// TIA Portal V17 export
// export: Created 2024-09-02T12:50:15.8804122Z, ExportSetting WithDefaults, DisplayName Totally Integrated Automation Portal, DisplayVersion V17, DisplayName TIA Portal Openness, DisplayVersion V17, DisplayName TIA Portal Version Control Interface, DisplayVersion V17, DisplayName STEP 7 Professional, DisplayVersion V17, DisplayName STEP 7 Safety, DisplayVersion V17, DisplayName WinCC Professional, DisplayVersion V17
FUNCTION "AnwFC_ZP_FunctionsSelection_OP70" : Void   // FC254, LAD
TITLE = function selections / Funktionsanwahlen
{ S7_Optimized_Access := 'TRUE' }
AUTHOR : OlegFuehrus
FAMILY : BA
NAME : BA
VERSION : 0.1
// stored: AutoNumber true, IsIECCheckEnabled false, SetENOAutomatically false, UDAEnableTagReadback false
   VAR_TEMP
      t_VKE0 : Bool;
      t_VKE1 : Bool;
      t_Enable_left : Bool;
      t_Enable_right : Bool;
      t_Fault : Bool;
      t_Function_left : Bool;
      t_Function_right : Bool;
      t_Line : Int;
      tBA_mode : Int;
   END_VAR
   VAR_TEMP   // added for the SCL form of the ladder/FBD networks
      _w1 : Bool;
      _w2 : Bool;
      _w3 : Bool;
      _w4 : Bool;
      _w5 : Bool;
   END_VAR
BEGIN

REGION Network 1: INIT
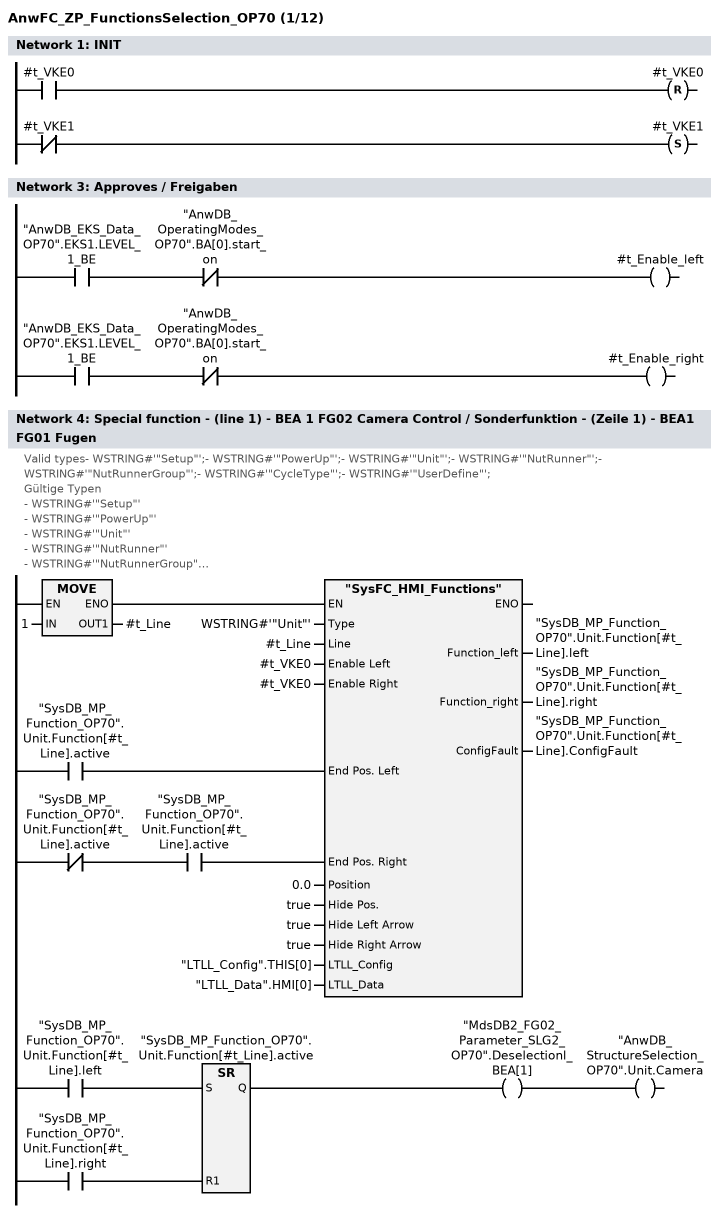
   RUNG wire#powerrail
      Contact( #t_VKE0 )
      R_Coil( #t_VKE0 )
   END_RUNG
   RUNG wire#powerrail
      I_Contact( #t_VKE1 )
      S_Coil( #t_VKE1 )
   END_RUNG
   // the same network as SCL:
   IF #t_VKE0 THEN #t_VKE0 := FALSE; END_IF;
   IF NOT #t_VKE1 THEN #t_VKE1 := TRUE; END_IF;
END_REGION

REGION Network 2: ######## UNIT ######### / ############ UNIT ############
END_REGION

REGION Network 3: Approves / Freigaben
   RUNG wire#powerrail
      Contact( "AnwDB_EKS_Data_OP70".EKS1.LEVEL_1_BE )
      I_Contact( "AnwDB_OperatingModes_OP70".BA[0].start_on )
      Coil( #t_Enable_left )
   END_RUNG
   RUNG wire#powerrail
      Contact( "AnwDB_EKS_Data_OP70".EKS1.LEVEL_1_BE )
      I_Contact( "AnwDB_OperatingModes_OP70".BA[0].start_on )
      Coil( #t_Enable_right )
   END_RUNG
   // the same network as SCL:
   #t_Enable_left := "AnwDB_EKS_Data_OP70".EKS1.LEVEL_1_BE AND NOT "AnwDB_OperatingModes_OP70".BA[0].start_on;
   #t_Enable_right := "AnwDB_EKS_Data_OP70".EKS1.LEVEL_1_BE AND NOT "AnwDB_OperatingModes_OP70".BA[0].start_on;
END_REGION

REGION Network 4: Special function - (line 1) - BEA 1 FG02 Camera Control / Sonderfunktion - (Zeile 1) - BEA1 FG01 Fugen
   // Valid types- WSTRING#'"Setup"';- WSTRING#'"PowerUp"';- WSTRING#'"Unit"';- WSTRING#'"NutRunner"';- WSTRING#'"NutRunnerGroup"';- WSTRING#'"CycleType"';- WSTRING#'"UserDefine"';
   // Gültige Typen
   // - WSTRING#'"Setup"'
   // - WSTRING#'"PowerUp"'
   // - WSTRING#'"Unit"'
   // - WSTRING#'"NutRunner"'
   // - WSTRING#'"NutRunnerGroup"'
   // - WSTRING#'"CycleType"'
   // - WSTRING#'"UserDefine"'
   RUNG wire#powerrail
      Move(in := 1, out1 => #t_Line)
      "SysFC_HMI_Functions"("End Pos. Left" := wire#w1, "End Pos. Right" := wire#w2, "Type" := WSTRING#'"Unit"', Line := #t_Line, "Enable Left" := #t_VKE0, "Enable Right" := #t_VKE0, Position := 0.0, "Hide Pos." := true, "Hide Left Arrow" := true, "Hide Right Arrow" := true, LTLL_Config := "LTLL_Config".THIS[0], LTLL_Data := "LTLL_Data".HMI[0], Function_left => "SysDB_MP_Function_OP70".Unit.Function[#t_Line].left, Function_right => "SysDB_MP_Function_OP70".Unit.Function[#t_Line].right, ConfigFault => "SysDB_MP_Function_OP70".Unit.Function[#t_Line].ConfigFault)
   END_RUNG
   RUNG wire#powerrail
      Contact( "SysDB_MP_Function_OP70".Unit.Function[#t_Line].active )
   END_RUNG wire#w1
   RUNG wire#powerrail
      I_Contact( "SysDB_MP_Function_OP70".Unit.Function[#t_Line].active )
      Contact( "SysDB_MP_Function_OP70".Unit.Function[#t_Line].active )
   END_RUNG wire#w2
   RUNG wire#powerrail
      Contact( "SysDB_MP_Function_OP70".Unit.Function[#t_Line].left )
      S_SR(operand := "SysDB_MP_Function_OP70".Unit.Function[#t_Line].active, r1 := wire#w3)
      Coil( "MdsDB2_FG02_Parameter_SLG2_OP70".Deselectionl_BEA[1] )
      Coil( "AnwDB_StructureSelection_OP70".Unit.Camera )
   END_RUNG
   RUNG wire#powerrail
      Contact( "SysDB_MP_Function_OP70".Unit.Function[#t_Line].right )
   END_RUNG wire#w3
   // the same network as SCL:
   #t_Line := 1;
   "SysFC_HMI_Functions"("Type" := WSTRING#'"Unit"',
                         Line := #t_Line,
                         "Enable Left" := #t_VKE0,
                         "Enable Right" := #t_VKE0,
                         "End Pos. Left" := "SysDB_MP_Function_OP70".Unit.Function[#t_Line].active,
                         "End Pos. Right" := NOT "SysDB_MP_Function_OP70".Unit.Function[#t_Line].active AND "SysDB_MP_Function_OP70".Unit.Function[#t_Line].active,
                         Position := 0.0,
                         "Hide Pos." := true,
                         "Hide Left Arrow" := true,
                         "Hide Right Arrow" := true,
                         LTLL_Config := "LTLL_Config".THIS[0],
                         LTLL_Data := "LTLL_Data".HMI[0],
                         Function_left => "SysDB_MP_Function_OP70".Unit.Function[#t_Line].left,
                         Function_right => "SysDB_MP_Function_OP70".Unit.Function[#t_Line].right,
                         ConfigFault => "SysDB_MP_Function_OP70".Unit.Function[#t_Line].ConfigFault);
   #_w1 := "SysDB_MP_Function_OP70".Unit.Function[#t_Line].right;
   IF "SysDB_MP_Function_OP70".Unit.Function[#t_Line].left THEN
       "SysDB_MP_Function_OP70".Unit.Function[#t_Line].active := TRUE;   // SR flip-flop
   END_IF;
   IF #_w1 THEN "SysDB_MP_Function_OP70".Unit.Function[#t_Line].active := FALSE; END_IF;
   "MdsDB2_FG02_Parameter_SLG2_OP70".Deselectionl_BEA[1] := "SysDB_MP_Function_OP70".Unit.Function[#t_Line].active;
   "AnwDB_StructureSelection_OP70".Unit.Camera := "SysDB_MP_Function_OP70".Unit.Function[#t_Line].active;
END_REGION

REGION Network 5: Special function - (line 2) - BEA 2 FG02 Replace plate / Sonderfunktion - (Zeile 1) - BEA1 FG01 Fugen
   // Valid types- WSTRING#'"Setup"';- WSTRING#'"PowerUp"';- WSTRING#'"Unit"';- WSTRING#'"NutRunner"';- WSTRING#'"NutRunnerGroup"';- WSTRING#'"CycleType"';- WSTRING#'"UserDefine"';
   // Gültige Typen
   // - WSTRING#'"Setup"'
   // - WSTRING#'"PowerUp"'
   // - WSTRING#'"Unit"'
   // - WSTRING#'"NutRunner"'
   // - WSTRING#'"NutRunnerGroup"'
   // - WSTRING#'"CycleType"'
   // - WSTRING#'"UserDefine"'
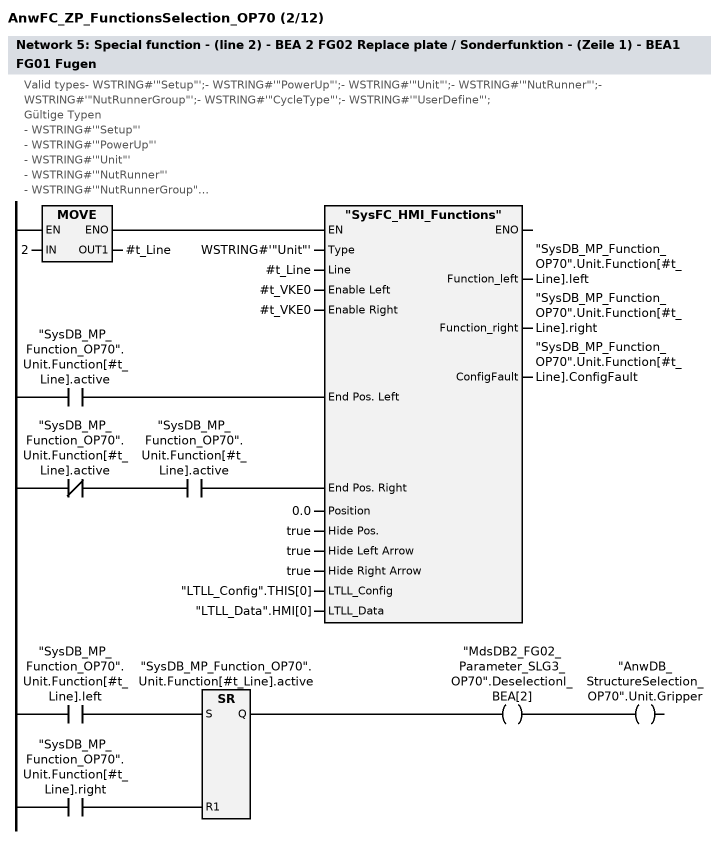
   RUNG wire#powerrail
      Move(in := 2, out1 => #t_Line)
      "SysFC_HMI_Functions"("End Pos. Left" := wire#w1, "End Pos. Right" := wire#w2, "Type" := WSTRING#'"Unit"', Line := #t_Line, "Enable Left" := #t_VKE0, "Enable Right" := #t_VKE0, Position := 0.0, "Hide Pos." := true, "Hide Left Arrow" := true, "Hide Right Arrow" := true, LTLL_Config := "LTLL_Config".THIS[0], LTLL_Data := "LTLL_Data".HMI[0], Function_left => "SysDB_MP_Function_OP70".Unit.Function[#t_Line].left, Function_right => "SysDB_MP_Function_OP70".Unit.Function[#t_Line].right, ConfigFault => "SysDB_MP_Function_OP70".Unit.Function[#t_Line].ConfigFault)
   END_RUNG
   RUNG wire#powerrail
      Contact( "SysDB_MP_Function_OP70".Unit.Function[#t_Line].active )
   END_RUNG wire#w1
   RUNG wire#powerrail
      I_Contact( "SysDB_MP_Function_OP70".Unit.Function[#t_Line].active )
      Contact( "SysDB_MP_Function_OP70".Unit.Function[#t_Line].active )
   END_RUNG wire#w2
   RUNG wire#powerrail
      Contact( "SysDB_MP_Function_OP70".Unit.Function[#t_Line].left )
      S_SR(operand := "SysDB_MP_Function_OP70".Unit.Function[#t_Line].active, r1 := wire#w3)
      Coil( "MdsDB2_FG02_Parameter_SLG3_OP70".Deselectionl_BEA[2] )
      Coil( "AnwDB_StructureSelection_OP70".Unit.Gripper )
   END_RUNG
   RUNG wire#powerrail
      Contact( "SysDB_MP_Function_OP70".Unit.Function[#t_Line].right )
   END_RUNG wire#w3
   // the same network as SCL:
   #t_Line := 2;
   "SysFC_HMI_Functions"("Type" := WSTRING#'"Unit"',
                         Line := #t_Line,
                         "Enable Left" := #t_VKE0,
                         "Enable Right" := #t_VKE0,
                         "End Pos. Left" := "SysDB_MP_Function_OP70".Unit.Function[#t_Line].active,
                         "End Pos. Right" := NOT "SysDB_MP_Function_OP70".Unit.Function[#t_Line].active AND "SysDB_MP_Function_OP70".Unit.Function[#t_Line].active,
                         Position := 0.0,
                         "Hide Pos." := true,
                         "Hide Left Arrow" := true,
                         "Hide Right Arrow" := true,
                         LTLL_Config := "LTLL_Config".THIS[0],
                         LTLL_Data := "LTLL_Data".HMI[0],
                         Function_left => "SysDB_MP_Function_OP70".Unit.Function[#t_Line].left,
                         Function_right => "SysDB_MP_Function_OP70".Unit.Function[#t_Line].right,
                         ConfigFault => "SysDB_MP_Function_OP70".Unit.Function[#t_Line].ConfigFault);
   #_w1 := "SysDB_MP_Function_OP70".Unit.Function[#t_Line].right;
   IF "SysDB_MP_Function_OP70".Unit.Function[#t_Line].left THEN
       "SysDB_MP_Function_OP70".Unit.Function[#t_Line].active := TRUE;   // SR flip-flop
   END_IF;
   IF #_w1 THEN "SysDB_MP_Function_OP70".Unit.Function[#t_Line].active := FALSE; END_IF;
   "MdsDB2_FG02_Parameter_SLG3_OP70".Deselectionl_BEA[2] := "SysDB_MP_Function_OP70".Unit.Function[#t_Line].active;
   "AnwDB_StructureSelection_OP70".Unit.Gripper := "SysDB_MP_Function_OP70".Unit.Function[#t_Line].active;
END_REGION

REGION Network 6: Special function - (line 3) - BEA 3 FG02 Screwdriver / Sonderfunktion - (Zeile 1) - BEA1 FG01 Fugen
   // Valid types- WSTRING#'"Setup"';- WSTRING#'"PowerUp"';- WSTRING#'"Unit"';- WSTRING#'"NutRunner"';- WSTRING#'"NutRunnerGroup"';- WSTRING#'"CycleType"';- WSTRING#'"UserDefine"';
   // Gültige Typen
   // - WSTRING#'"Setup"'
   // - WSTRING#'"PowerUp"'
   // - WSTRING#'"Unit"'
   // - WSTRING#'"NutRunner"'
   // - WSTRING#'"NutRunnerGroup"'
   // - WSTRING#'"CycleType"'
   // - WSTRING#'"UserDefine"'
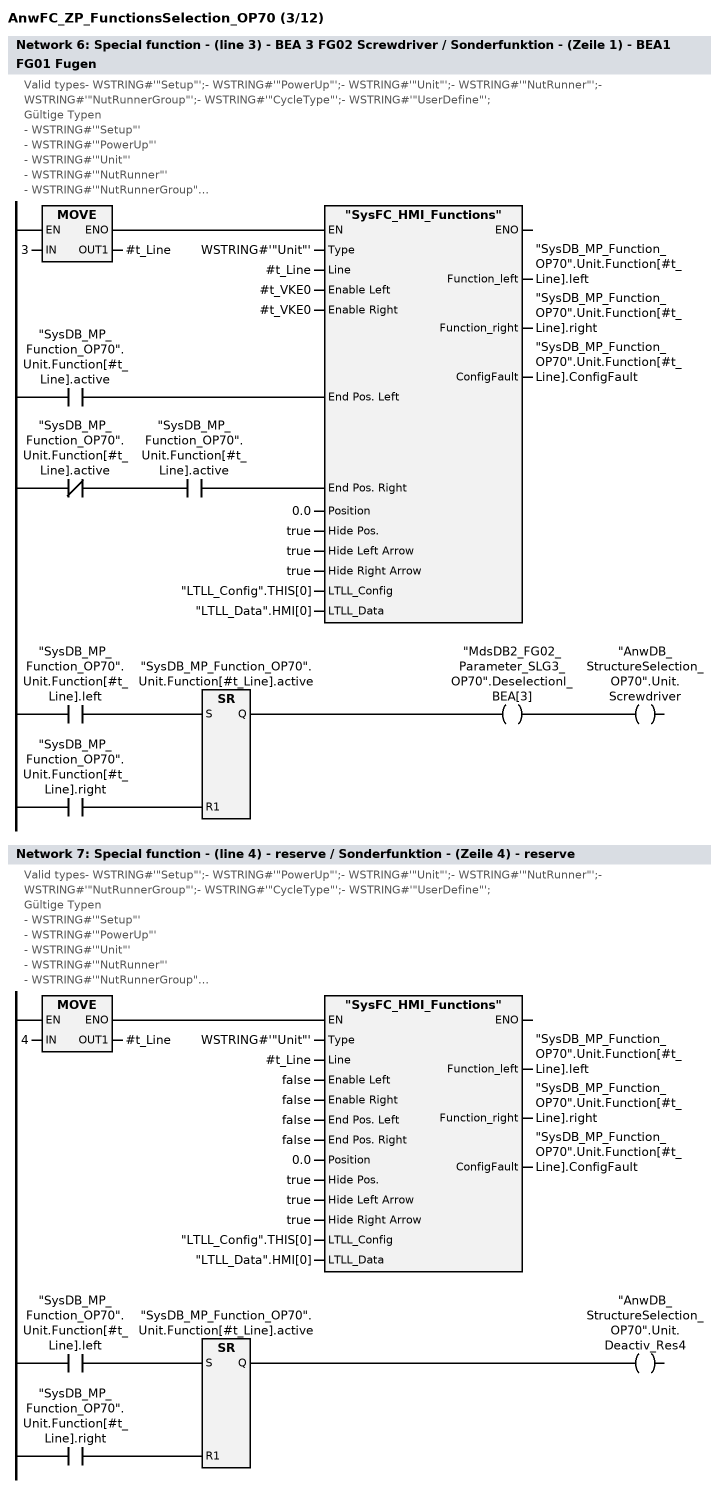
   RUNG wire#powerrail
      Move(in := 3, out1 => #t_Line)
      "SysFC_HMI_Functions"("End Pos. Left" := wire#w1, "End Pos. Right" := wire#w2, "Type" := WSTRING#'"Unit"', Line := #t_Line, "Enable Left" := #t_VKE0, "Enable Right" := #t_VKE0, Position := 0.0, "Hide Pos." := true, "Hide Left Arrow" := true, "Hide Right Arrow" := true, LTLL_Config := "LTLL_Config".THIS[0], LTLL_Data := "LTLL_Data".HMI[0], Function_left => "SysDB_MP_Function_OP70".Unit.Function[#t_Line].left, Function_right => "SysDB_MP_Function_OP70".Unit.Function[#t_Line].right, ConfigFault => "SysDB_MP_Function_OP70".Unit.Function[#t_Line].ConfigFault)
   END_RUNG
   RUNG wire#powerrail
      Contact( "SysDB_MP_Function_OP70".Unit.Function[#t_Line].active )
   END_RUNG wire#w1
   RUNG wire#powerrail
      I_Contact( "SysDB_MP_Function_OP70".Unit.Function[#t_Line].active )
      Contact( "SysDB_MP_Function_OP70".Unit.Function[#t_Line].active )
   END_RUNG wire#w2
   RUNG wire#powerrail
      Contact( "SysDB_MP_Function_OP70".Unit.Function[#t_Line].left )
      S_SR(operand := "SysDB_MP_Function_OP70".Unit.Function[#t_Line].active, r1 := wire#w3)
      Coil( "MdsDB2_FG02_Parameter_SLG3_OP70".Deselectionl_BEA[3] )
      Coil( "AnwDB_StructureSelection_OP70".Unit.Screwdriver )
   END_RUNG
   RUNG wire#powerrail
      Contact( "SysDB_MP_Function_OP70".Unit.Function[#t_Line].right )
   END_RUNG wire#w3
   // the same network as SCL:
   #t_Line := 3;
   "SysFC_HMI_Functions"("Type" := WSTRING#'"Unit"',
                         Line := #t_Line,
                         "Enable Left" := #t_VKE0,
                         "Enable Right" := #t_VKE0,
                         "End Pos. Left" := "SysDB_MP_Function_OP70".Unit.Function[#t_Line].active,
                         "End Pos. Right" := NOT "SysDB_MP_Function_OP70".Unit.Function[#t_Line].active AND "SysDB_MP_Function_OP70".Unit.Function[#t_Line].active,
                         Position := 0.0,
                         "Hide Pos." := true,
                         "Hide Left Arrow" := true,
                         "Hide Right Arrow" := true,
                         LTLL_Config := "LTLL_Config".THIS[0],
                         LTLL_Data := "LTLL_Data".HMI[0],
                         Function_left => "SysDB_MP_Function_OP70".Unit.Function[#t_Line].left,
                         Function_right => "SysDB_MP_Function_OP70".Unit.Function[#t_Line].right,
                         ConfigFault => "SysDB_MP_Function_OP70".Unit.Function[#t_Line].ConfigFault);
   #_w1 := "SysDB_MP_Function_OP70".Unit.Function[#t_Line].right;
   IF "SysDB_MP_Function_OP70".Unit.Function[#t_Line].left THEN
       "SysDB_MP_Function_OP70".Unit.Function[#t_Line].active := TRUE;   // SR flip-flop
   END_IF;
   IF #_w1 THEN "SysDB_MP_Function_OP70".Unit.Function[#t_Line].active := FALSE; END_IF;
   "MdsDB2_FG02_Parameter_SLG3_OP70".Deselectionl_BEA[3] := "SysDB_MP_Function_OP70".Unit.Function[#t_Line].active;
   "AnwDB_StructureSelection_OP70".Unit.Screwdriver := "SysDB_MP_Function_OP70".Unit.Function[#t_Line].active;
END_REGION

REGION Network 7: Special function - (line 4) - reserve / Sonderfunktion - (Zeile 4) - reserve
   // Valid types- WSTRING#'"Setup"';- WSTRING#'"PowerUp"';- WSTRING#'"Unit"';- WSTRING#'"NutRunner"';- WSTRING#'"NutRunnerGroup"';- WSTRING#'"CycleType"';- WSTRING#'"UserDefine"';
   // Gültige Typen
   // - WSTRING#'"Setup"'
   // - WSTRING#'"PowerUp"'
   // - WSTRING#'"Unit"'
   // - WSTRING#'"NutRunner"'
   // - WSTRING#'"NutRunnerGroup"'
   // - WSTRING#'"CycleType"'
   // - WSTRING#'"UserDefine"'
   RUNG wire#powerrail
      Move(in := 4, out1 => #t_Line)
      "SysFC_HMI_Functions"("Type" := WSTRING#'"Unit"', Line := #t_Line, "Enable Left" := false, "Enable Right" := false, "End Pos. Left" := false, "End Pos. Right" := false, Position := 0.0, "Hide Pos." := true, "Hide Left Arrow" := true, "Hide Right Arrow" := true, LTLL_Config := "LTLL_Config".THIS[0], LTLL_Data := "LTLL_Data".HMI[0], Function_left => "SysDB_MP_Function_OP70".Unit.Function[#t_Line].left, Function_right => "SysDB_MP_Function_OP70".Unit.Function[#t_Line].right, ConfigFault => "SysDB_MP_Function_OP70".Unit.Function[#t_Line].ConfigFault)
   END_RUNG
   RUNG wire#powerrail
      Contact( "SysDB_MP_Function_OP70".Unit.Function[#t_Line].left )
      S_SR(operand := "SysDB_MP_Function_OP70".Unit.Function[#t_Line].active, r1 := wire#w1)
      Coil( "AnwDB_StructureSelection_OP70".Unit.Deactiv_Res4 )
   END_RUNG
   RUNG wire#powerrail
      Contact( "SysDB_MP_Function_OP70".Unit.Function[#t_Line].right )
   END_RUNG wire#w1
   // the same network as SCL:
   #t_Line := 4;
   "SysFC_HMI_Functions"("Type" := WSTRING#'"Unit"',
                         Line := #t_Line,
                         "Enable Left" := false,
                         "Enable Right" := false,
                         "End Pos. Left" := false,
                         "End Pos. Right" := false,
                         Position := 0.0,
                         "Hide Pos." := true,
                         "Hide Left Arrow" := true,
                         "Hide Right Arrow" := true,
                         LTLL_Config := "LTLL_Config".THIS[0],
                         LTLL_Data := "LTLL_Data".HMI[0],
                         Function_left => "SysDB_MP_Function_OP70".Unit.Function[#t_Line].left,
                         Function_right => "SysDB_MP_Function_OP70".Unit.Function[#t_Line].right,
                         ConfigFault => "SysDB_MP_Function_OP70".Unit.Function[#t_Line].ConfigFault);
   #_w1 := "SysDB_MP_Function_OP70".Unit.Function[#t_Line].right;
   IF "SysDB_MP_Function_OP70".Unit.Function[#t_Line].left THEN
       "SysDB_MP_Function_OP70".Unit.Function[#t_Line].active := TRUE;   // SR flip-flop
   END_IF;
   IF #_w1 THEN "SysDB_MP_Function_OP70".Unit.Function[#t_Line].active := FALSE; END_IF;
   "AnwDB_StructureSelection_OP70".Unit.Deactiv_Res4 := "SysDB_MP_Function_OP70".Unit.Function[#t_Line].active;
END_REGION

REGION Network 8: Special function - (line 5) - reserve / Sonderfunktion - (Zeile 5) - reserve
   // Valid types- WSTRING#'"Setup"';- WSTRING#'"PowerUp"';- WSTRING#'"Unit"';- WSTRING#'"NutRunner"';- WSTRING#'"NutRunnerGroup"';- WSTRING#'"CycleType"';- WSTRING#'"UserDefine"';
   // Gültige Typen
   // - WSTRING#'"Setup"'
   // - WSTRING#'"PowerUp"'
   // - WSTRING#'"Unit"'
   // - WSTRING#'"NutRunner"'
   // - WSTRING#'"NutRunnerGroup"'
   // - WSTRING#'"CycleType"'
   // - WSTRING#'"UserDefine"'
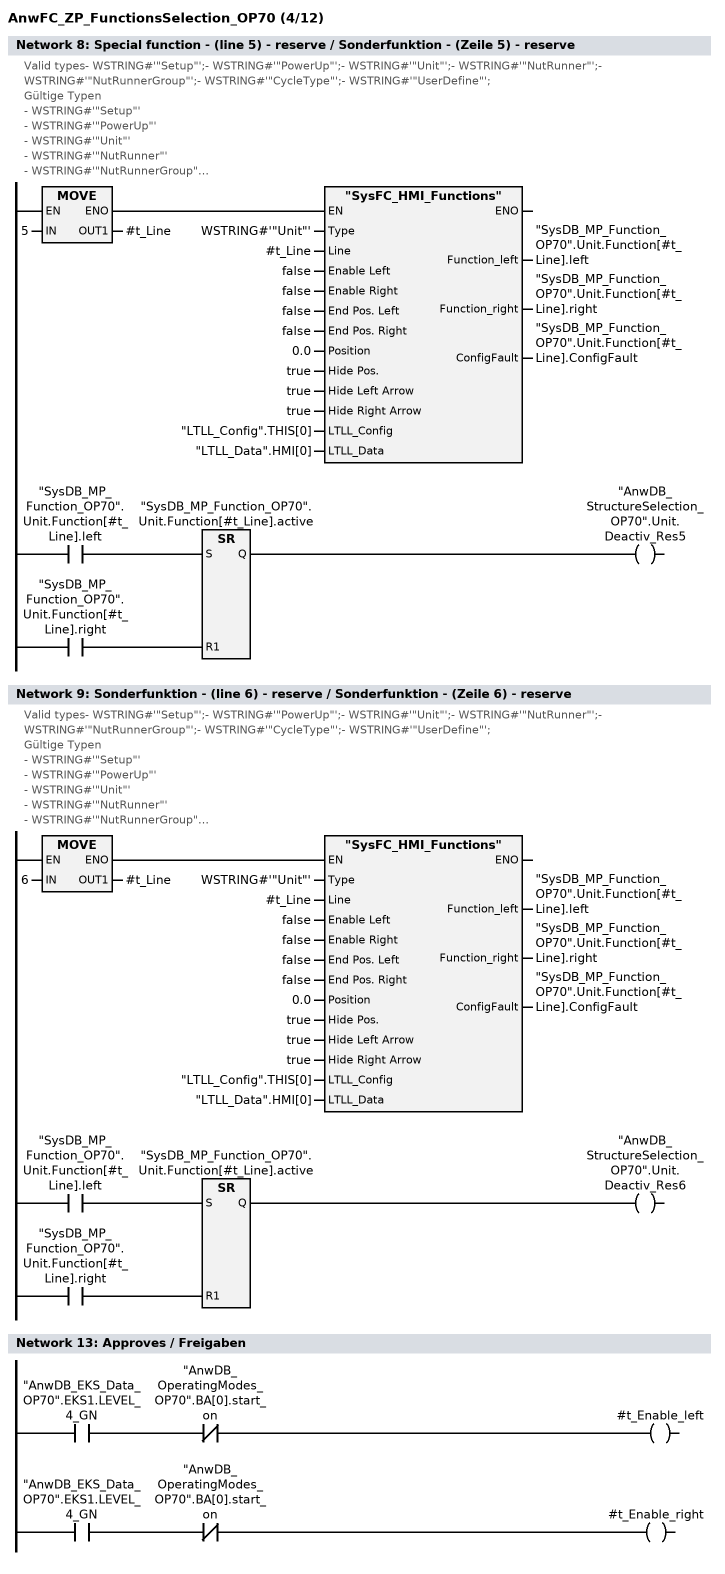
   RUNG wire#powerrail
      Move(in := 5, out1 => #t_Line)
      "SysFC_HMI_Functions"("Type" := WSTRING#'"Unit"', Line := #t_Line, "Enable Left" := false, "Enable Right" := false, "End Pos. Left" := false, "End Pos. Right" := false, Position := 0.0, "Hide Pos." := true, "Hide Left Arrow" := true, "Hide Right Arrow" := true, LTLL_Config := "LTLL_Config".THIS[0], LTLL_Data := "LTLL_Data".HMI[0], Function_left => "SysDB_MP_Function_OP70".Unit.Function[#t_Line].left, Function_right => "SysDB_MP_Function_OP70".Unit.Function[#t_Line].right, ConfigFault => "SysDB_MP_Function_OP70".Unit.Function[#t_Line].ConfigFault)
   END_RUNG
   RUNG wire#powerrail
      Contact( "SysDB_MP_Function_OP70".Unit.Function[#t_Line].left )
      S_SR(operand := "SysDB_MP_Function_OP70".Unit.Function[#t_Line].active, r1 := wire#w1)
      Coil( "AnwDB_StructureSelection_OP70".Unit.Deactiv_Res5 )
   END_RUNG
   RUNG wire#powerrail
      Contact( "SysDB_MP_Function_OP70".Unit.Function[#t_Line].right )
   END_RUNG wire#w1
   // the same network as SCL:
   #t_Line := 5;
   "SysFC_HMI_Functions"("Type" := WSTRING#'"Unit"',
                         Line := #t_Line,
                         "Enable Left" := false,
                         "Enable Right" := false,
                         "End Pos. Left" := false,
                         "End Pos. Right" := false,
                         Position := 0.0,
                         "Hide Pos." := true,
                         "Hide Left Arrow" := true,
                         "Hide Right Arrow" := true,
                         LTLL_Config := "LTLL_Config".THIS[0],
                         LTLL_Data := "LTLL_Data".HMI[0],
                         Function_left => "SysDB_MP_Function_OP70".Unit.Function[#t_Line].left,
                         Function_right => "SysDB_MP_Function_OP70".Unit.Function[#t_Line].right,
                         ConfigFault => "SysDB_MP_Function_OP70".Unit.Function[#t_Line].ConfigFault);
   #_w1 := "SysDB_MP_Function_OP70".Unit.Function[#t_Line].right;
   IF "SysDB_MP_Function_OP70".Unit.Function[#t_Line].left THEN
       "SysDB_MP_Function_OP70".Unit.Function[#t_Line].active := TRUE;   // SR flip-flop
   END_IF;
   IF #_w1 THEN "SysDB_MP_Function_OP70".Unit.Function[#t_Line].active := FALSE; END_IF;
   "AnwDB_StructureSelection_OP70".Unit.Deactiv_Res5 := "SysDB_MP_Function_OP70".Unit.Function[#t_Line].active;
END_REGION

REGION Network 9: Sonderfunktion - (line 6) - reserve / Sonderfunktion - (Zeile 6) - reserve
   // Valid types- WSTRING#'"Setup"';- WSTRING#'"PowerUp"';- WSTRING#'"Unit"';- WSTRING#'"NutRunner"';- WSTRING#'"NutRunnerGroup"';- WSTRING#'"CycleType"';- WSTRING#'"UserDefine"';
   // Gültige Typen
   // - WSTRING#'"Setup"'
   // - WSTRING#'"PowerUp"'
   // - WSTRING#'"Unit"'
   // - WSTRING#'"NutRunner"'
   // - WSTRING#'"NutRunnerGroup"'
   // - WSTRING#'"CycleType"'
   // - WSTRING#'"UserDefine"'
   RUNG wire#powerrail
      Move(in := 6, out1 => #t_Line)
      "SysFC_HMI_Functions"("Type" := WSTRING#'"Unit"', Line := #t_Line, "Enable Left" := false, "Enable Right" := false, "End Pos. Left" := false, "End Pos. Right" := false, Position := 0.0, "Hide Pos." := true, "Hide Left Arrow" := true, "Hide Right Arrow" := true, LTLL_Config := "LTLL_Config".THIS[0], LTLL_Data := "LTLL_Data".HMI[0], Function_left => "SysDB_MP_Function_OP70".Unit.Function[#t_Line].left, Function_right => "SysDB_MP_Function_OP70".Unit.Function[#t_Line].right, ConfigFault => "SysDB_MP_Function_OP70".Unit.Function[#t_Line].ConfigFault)
   END_RUNG
   RUNG wire#powerrail
      Contact( "SysDB_MP_Function_OP70".Unit.Function[#t_Line].left )
      S_SR(operand := "SysDB_MP_Function_OP70".Unit.Function[#t_Line].active, r1 := wire#w1)
      Coil( "AnwDB_StructureSelection_OP70".Unit.Deactiv_Res6 )
   END_RUNG
   RUNG wire#powerrail
      Contact( "SysDB_MP_Function_OP70".Unit.Function[#t_Line].right )
   END_RUNG wire#w1
   // the same network as SCL:
   #t_Line := 6;
   "SysFC_HMI_Functions"("Type" := WSTRING#'"Unit"',
                         Line := #t_Line,
                         "Enable Left" := false,
                         "Enable Right" := false,
                         "End Pos. Left" := false,
                         "End Pos. Right" := false,
                         Position := 0.0,
                         "Hide Pos." := true,
                         "Hide Left Arrow" := true,
                         "Hide Right Arrow" := true,
                         LTLL_Config := "LTLL_Config".THIS[0],
                         LTLL_Data := "LTLL_Data".HMI[0],
                         Function_left => "SysDB_MP_Function_OP70".Unit.Function[#t_Line].left,
                         Function_right => "SysDB_MP_Function_OP70".Unit.Function[#t_Line].right,
                         ConfigFault => "SysDB_MP_Function_OP70".Unit.Function[#t_Line].ConfigFault);
   #_w1 := "SysDB_MP_Function_OP70".Unit.Function[#t_Line].right;
   IF "SysDB_MP_Function_OP70".Unit.Function[#t_Line].left THEN
       "SysDB_MP_Function_OP70".Unit.Function[#t_Line].active := TRUE;   // SR flip-flop
   END_IF;
   IF #_w1 THEN "SysDB_MP_Function_OP70".Unit.Function[#t_Line].active := FALSE; END_IF;
   "AnwDB_StructureSelection_OP70".Unit.Deactiv_Res6 := "SysDB_MP_Function_OP70".Unit.Function[#t_Line].active;
END_REGION

REGION Network 10: ######## NUT RUNNER ######### / ############ NUT RUNNER ############
END_REGION

REGION Network 11: ######## NUT RUNNER GROUP ######### / ############ NUT RUNNER GROUP ############
END_REGION

REGION Network 12: ######## CYCLE TYPE ######### / ############ CYCLE TYPE ############
END_REGION

REGION Network 13: Approves / Freigaben
   RUNG wire#powerrail
      Contact( "AnwDB_EKS_Data_OP70".EKS1.LEVEL_4_GN )
      I_Contact( "AnwDB_OperatingModes_OP70".BA[0].start_on )
      Coil( #t_Enable_left )
   END_RUNG
   RUNG wire#powerrail
      Contact( "AnwDB_EKS_Data_OP70".EKS1.LEVEL_4_GN )
      I_Contact( "AnwDB_OperatingModes_OP70".BA[0].start_on )
      Coil( #t_Enable_right )
   END_RUNG
   // the same network as SCL:
   #t_Enable_left := "AnwDB_EKS_Data_OP70".EKS1.LEVEL_4_GN AND NOT "AnwDB_OperatingModes_OP70".BA[0].start_on;
   #t_Enable_right := "AnwDB_EKS_Data_OP70".EKS1.LEVEL_4_GN AND NOT "AnwDB_OperatingModes_OP70".BA[0].start_on;
END_REGION

REGION Network 14: CycleType - (line 1) - Single step mode / CycleType - (Zeile 1) - Einzelschritt
   // Valid types- WSTRING#'"Setup"';- WSTRING#'"PowerUp"';- WSTRING#'"Unit"';- WSTRING#'"NutRunner"';- WSTRING#'"NutRunnerGroup"';- WSTRING#'"CycleType"';- WSTRING#'"UserDefine"';
   // Gültige Typen
   // - WSTRING#'"Setup"'
   // - WSTRING#'"PowerUp"'
   // - WSTRING#'"Unit"'
   // - WSTRING#'"NutRunner"'
   // - WSTRING#'"NutRunnerGroup"'
   // - WSTRING#'"CycleType"'
   // - WSTRING#'"UserDefine"'
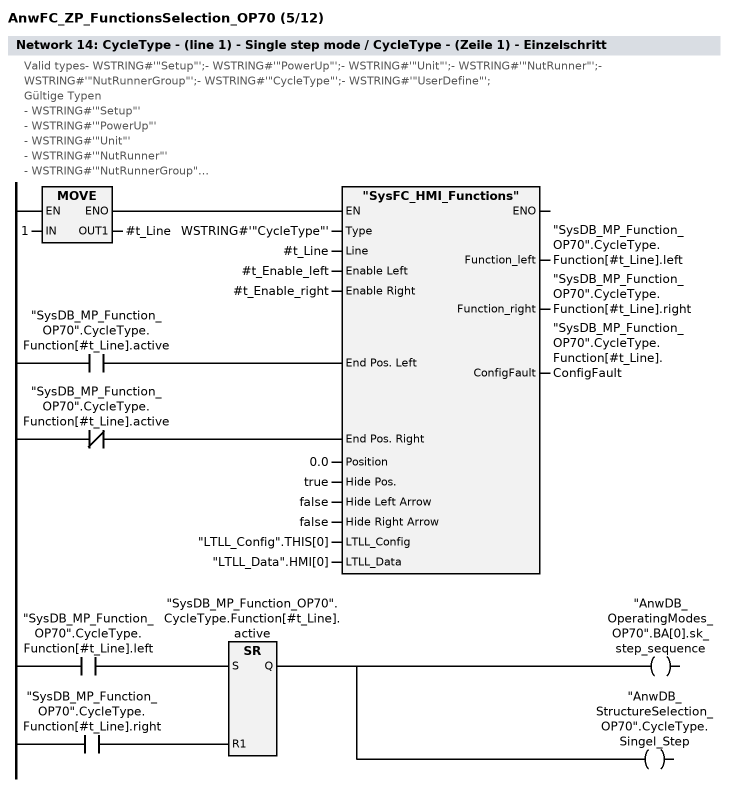
   RUNG wire#powerrail
      Move(in := 1, out1 => #t_Line)
      "SysFC_HMI_Functions"("End Pos. Left" := wire#w1, "End Pos. Right" := wire#w2, "Type" := WSTRING#'"CycleType"', Line := #t_Line, "Enable Left" := #t_Enable_left, "Enable Right" := #t_Enable_right, Position := 0.0, "Hide Pos." := true, "Hide Left Arrow" := false, "Hide Right Arrow" := false, LTLL_Config := "LTLL_Config".THIS[0], LTLL_Data := "LTLL_Data".HMI[0], Function_left => "SysDB_MP_Function_OP70".CycleType.Function[#t_Line].left, Function_right => "SysDB_MP_Function_OP70".CycleType.Function[#t_Line].right, ConfigFault => "SysDB_MP_Function_OP70".CycleType.Function[#t_Line].ConfigFault)
   END_RUNG
   RUNG wire#powerrail
      Contact( "SysDB_MP_Function_OP70".CycleType.Function[#t_Line].active )
   END_RUNG wire#w1
   RUNG wire#powerrail
      I_Contact( "SysDB_MP_Function_OP70".CycleType.Function[#t_Line].active )
   END_RUNG wire#w2
   RUNG wire#powerrail
      Contact( "SysDB_MP_Function_OP70".CycleType.Function[#t_Line].left )
      S_SR(operand := "SysDB_MP_Function_OP70".CycleType.Function[#t_Line].active, r1 := wire#w3)
      wire#w4
      Coil( "AnwDB_OperatingModes_OP70".BA[0].sk_step_sequence )
   END_RUNG
   RUNG wire#powerrail
      Contact( "SysDB_MP_Function_OP70".CycleType.Function[#t_Line].right )
   END_RUNG wire#w3
   RUNG wire#w4
      Coil( "AnwDB_StructureSelection_OP70".CycleType.Singel_Step )
   END_RUNG
   // the same network as SCL:
   #t_Line := 1;
   "SysFC_HMI_Functions"("Type" := WSTRING#'"CycleType"',
                         Line := #t_Line,
                         "Enable Left" := #t_Enable_left,
                         "Enable Right" := #t_Enable_right,
                         "End Pos. Left" := "SysDB_MP_Function_OP70".CycleType.Function[#t_Line].active,
                         "End Pos. Right" := NOT "SysDB_MP_Function_OP70".CycleType.Function[#t_Line].active,
                         Position := 0.0,
                         "Hide Pos." := true,
                         "Hide Left Arrow" := false,
                         "Hide Right Arrow" := false,
                         LTLL_Config := "LTLL_Config".THIS[0],
                         LTLL_Data := "LTLL_Data".HMI[0],
                         Function_left => "SysDB_MP_Function_OP70".CycleType.Function[#t_Line].left,
                         Function_right => "SysDB_MP_Function_OP70".CycleType.Function[#t_Line].right,
                         ConfigFault => "SysDB_MP_Function_OP70".CycleType.Function[#t_Line].ConfigFault);
   #_w1 := "SysDB_MP_Function_OP70".CycleType.Function[#t_Line].right;
   IF "SysDB_MP_Function_OP70".CycleType.Function[#t_Line].left THEN
       "SysDB_MP_Function_OP70".CycleType.Function[#t_Line].active := TRUE;   // SR flip-flop
   END_IF;
   IF #_w1 THEN "SysDB_MP_Function_OP70".CycleType.Function[#t_Line].active := FALSE; END_IF;
   "AnwDB_OperatingModes_OP70".BA[0].sk_step_sequence := "SysDB_MP_Function_OP70".CycleType.Function[#t_Line].active;
   "AnwDB_StructureSelection_OP70".CycleType.Singel_Step := "SysDB_MP_Function_OP70".CycleType.Function[#t_Line].active;
END_REGION

REGION Network 15: CycleType - (line 2) - Service / CycleType - (Zeile 2) - Service
   // Valid types- WSTRING#'"Setup"';- WSTRING#'"PowerUp"';- WSTRING#'"Unit"';- WSTRING#'"NutRunner"';- WSTRING#'"NutRunnerGroup"';- WSTRING#'"CycleType"';- WSTRING#'"UserDefine"';
   // Gültige Typen
   // - WSTRING#'"Setup"'
   // - WSTRING#'"PowerUp"'
   // - WSTRING#'"Unit"'
   // - WSTRING#'"NutRunner"'
   // - WSTRING#'"NutRunnerGroup"'
   // - WSTRING#'"CycleType"'
   // - WSTRING#'"UserDefine"'
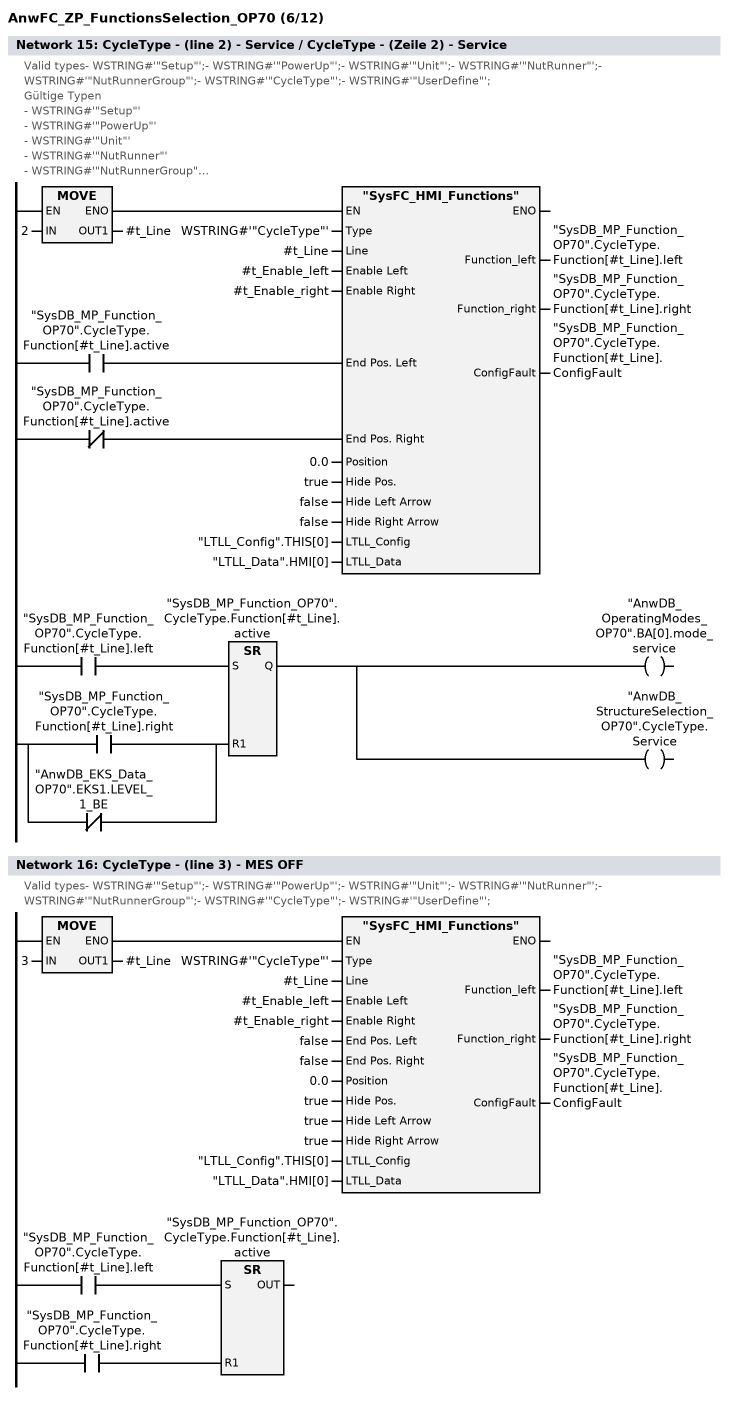
   RUNG wire#powerrail
      Move(in := 2, out1 => #t_Line)
      "SysFC_HMI_Functions"("End Pos. Left" := wire#w1, "End Pos. Right" := wire#w2, "Type" := WSTRING#'"CycleType"', Line := #t_Line, "Enable Left" := #t_Enable_left, "Enable Right" := #t_Enable_right, Position := 0.0, "Hide Pos." := true, "Hide Left Arrow" := false, "Hide Right Arrow" := false, LTLL_Config := "LTLL_Config".THIS[0], LTLL_Data := "LTLL_Data".HMI[0], Function_left => "SysDB_MP_Function_OP70".CycleType.Function[#t_Line].left, Function_right => "SysDB_MP_Function_OP70".CycleType.Function[#t_Line].right, ConfigFault => "SysDB_MP_Function_OP70".CycleType.Function[#t_Line].ConfigFault)
   END_RUNG
   RUNG wire#powerrail
      Contact( "SysDB_MP_Function_OP70".CycleType.Function[#t_Line].active )
   END_RUNG wire#w1
   RUNG wire#powerrail
      I_Contact( "SysDB_MP_Function_OP70".CycleType.Function[#t_Line].active )
   END_RUNG wire#w2
   RUNG wire#powerrail
      Contact( "SysDB_MP_Function_OP70".CycleType.Function[#t_Line].left )
      S_SR(operand := "SysDB_MP_Function_OP70".CycleType.Function[#t_Line].active, r1 := wire#w3)
      wire#w4
      Coil( "AnwDB_OperatingModes_OP70".BA[0].mode_service )
   END_RUNG
   RUNG wire#powerrail
      Contact( "SysDB_MP_Function_OP70".CycleType.Function[#t_Line].right )
   END_RUNG wire#w3
   RUNG wire#powerrail
      I_Contact( "AnwDB_EKS_Data_OP70".EKS1.LEVEL_1_BE )
   END_RUNG wire#w3
   RUNG wire#w4
      Coil( "AnwDB_StructureSelection_OP70".CycleType.Service )
   END_RUNG
   // the same network as SCL:
   #t_Line := 2;
   "SysFC_HMI_Functions"("Type" := WSTRING#'"CycleType"',
                         Line := #t_Line,
                         "Enable Left" := #t_Enable_left,
                         "Enable Right" := #t_Enable_right,
                         "End Pos. Left" := "SysDB_MP_Function_OP70".CycleType.Function[#t_Line].active,
                         "End Pos. Right" := NOT "SysDB_MP_Function_OP70".CycleType.Function[#t_Line].active,
                         Position := 0.0,
                         "Hide Pos." := true,
                         "Hide Left Arrow" := false,
                         "Hide Right Arrow" := false,
                         LTLL_Config := "LTLL_Config".THIS[0],
                         LTLL_Data := "LTLL_Data".HMI[0],
                         Function_left => "SysDB_MP_Function_OP70".CycleType.Function[#t_Line].left,
                         Function_right => "SysDB_MP_Function_OP70".CycleType.Function[#t_Line].right,
                         ConfigFault => "SysDB_MP_Function_OP70".CycleType.Function[#t_Line].ConfigFault);
   #_w1 := "SysDB_MP_Function_OP70".CycleType.Function[#t_Line].right OR NOT "AnwDB_EKS_Data_OP70".EKS1.LEVEL_1_BE;
   IF "SysDB_MP_Function_OP70".CycleType.Function[#t_Line].left THEN
       "SysDB_MP_Function_OP70".CycleType.Function[#t_Line].active := TRUE;   // SR flip-flop
   END_IF;
   IF #_w1 THEN "SysDB_MP_Function_OP70".CycleType.Function[#t_Line].active := FALSE; END_IF;
   "AnwDB_OperatingModes_OP70".BA[0].mode_service := "SysDB_MP_Function_OP70".CycleType.Function[#t_Line].active;
   "AnwDB_StructureSelection_OP70".CycleType.Service := "SysDB_MP_Function_OP70".CycleType.Function[#t_Line].active;
END_REGION

REGION Network 16: CycleType - (line 3) - MES OFF
   // Valid types- WSTRING#'"Setup"';- WSTRING#'"PowerUp"';- WSTRING#'"Unit"';- WSTRING#'"NutRunner"';- WSTRING#'"NutRunnerGroup"';- WSTRING#'"CycleType"';- WSTRING#'"UserDefine"';
   RUNG wire#powerrail
      Move(in := 3, out1 => #t_Line)
      "SysFC_HMI_Functions"("Type" := WSTRING#'"CycleType"', Line := #t_Line, "Enable Left" := #t_Enable_left, "Enable Right" := #t_Enable_right, "End Pos. Left" := false, "End Pos. Right" := false, Position := 0.0, "Hide Pos." := true, "Hide Left Arrow" := true, "Hide Right Arrow" := true, LTLL_Config := "LTLL_Config".THIS[0], LTLL_Data := "LTLL_Data".HMI[0], Function_left => "SysDB_MP_Function_OP70".CycleType.Function[#t_Line].left, Function_right => "SysDB_MP_Function_OP70".CycleType.Function[#t_Line].right, ConfigFault => "SysDB_MP_Function_OP70".CycleType.Function[#t_Line].ConfigFault)
   END_RUNG
   RUNG wire#powerrail
      Contact( "SysDB_MP_Function_OP70".CycleType.Function[#t_Line].left )
      S_SR(operand := "SysDB_MP_Function_OP70".CycleType.Function[#t_Line].active, r1 := wire#w1)
   END_RUNG
   RUNG wire#powerrail
      Contact( "SysDB_MP_Function_OP70".CycleType.Function[#t_Line].right )
   END_RUNG wire#w1
   // the same network as SCL:
   #t_Line := 3;
   "SysFC_HMI_Functions"("Type" := WSTRING#'"CycleType"',
                         Line := #t_Line,
                         "Enable Left" := #t_Enable_left,
                         "Enable Right" := #t_Enable_right,
                         "End Pos. Left" := false,
                         "End Pos. Right" := false,
                         Position := 0.0,
                         "Hide Pos." := true,
                         "Hide Left Arrow" := true,
                         "Hide Right Arrow" := true,
                         LTLL_Config := "LTLL_Config".THIS[0],
                         LTLL_Data := "LTLL_Data".HMI[0],
                         Function_left => "SysDB_MP_Function_OP70".CycleType.Function[#t_Line].left,
                         Function_right => "SysDB_MP_Function_OP70".CycleType.Function[#t_Line].right,
                         ConfigFault => "SysDB_MP_Function_OP70".CycleType.Function[#t_Line].ConfigFault);
   #_w1 := "SysDB_MP_Function_OP70".CycleType.Function[#t_Line].right;
   IF "SysDB_MP_Function_OP70".CycleType.Function[#t_Line].left THEN
       "SysDB_MP_Function_OP70".CycleType.Function[#t_Line].active := TRUE;   // SR flip-flop
   END_IF;
   IF #_w1 THEN "SysDB_MP_Function_OP70".CycleType.Function[#t_Line].active := FALSE; END_IF;
END_REGION

REGION Network 17: CycleType - (line 4) - Damper Cap Feeding Bypass
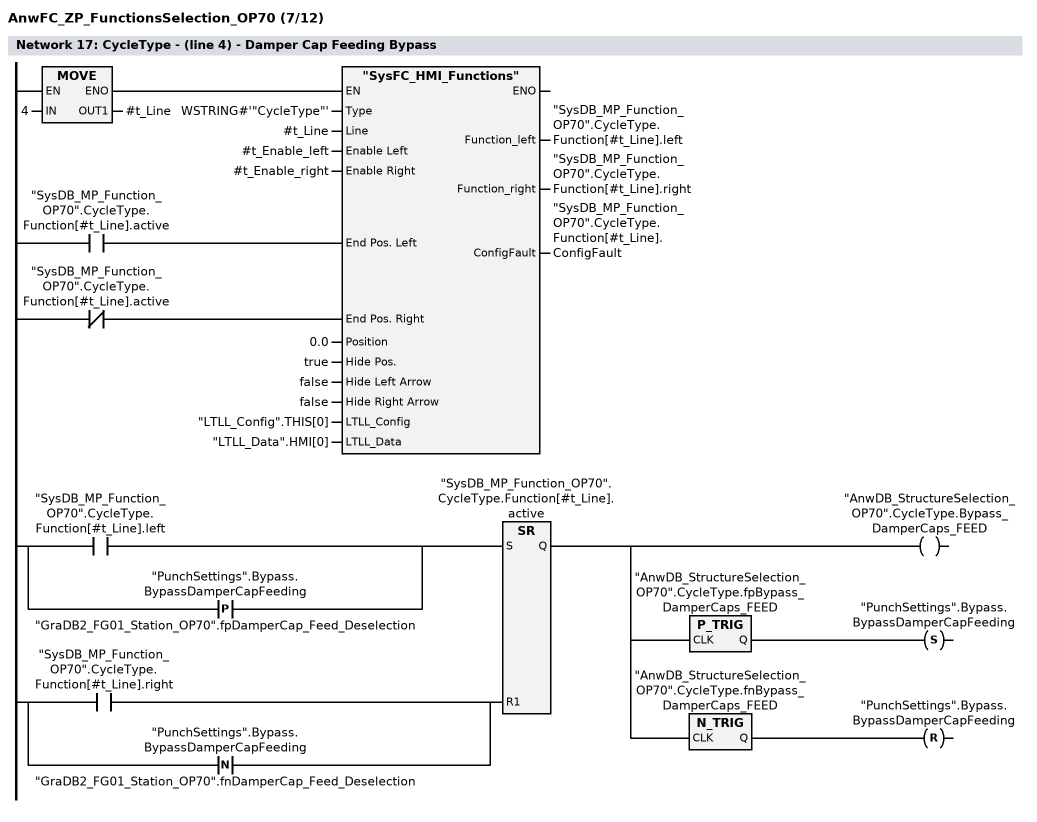
   RUNG wire#powerrail
      Move(in := 4, out1 => #t_Line)
      "SysFC_HMI_Functions"("End Pos. Left" := wire#w1, "End Pos. Right" := wire#w2, "Type" := WSTRING#'"CycleType"', Line := #t_Line, "Enable Left" := #t_Enable_left, "Enable Right" := #t_Enable_right, Position := 0.0, "Hide Pos." := true, "Hide Left Arrow" := false, "Hide Right Arrow" := false, LTLL_Config := "LTLL_Config".THIS[0], LTLL_Data := "LTLL_Data".HMI[0], Function_left => "SysDB_MP_Function_OP70".CycleType.Function[#t_Line].left, Function_right => "SysDB_MP_Function_OP70".CycleType.Function[#t_Line].right, ConfigFault => "SysDB_MP_Function_OP70".CycleType.Function[#t_Line].ConfigFault)
   END_RUNG
   RUNG wire#powerrail
      Contact( "SysDB_MP_Function_OP70".CycleType.Function[#t_Line].active )
   END_RUNG wire#w1
   RUNG wire#powerrail
      I_Contact( "SysDB_MP_Function_OP70".CycleType.Function[#t_Line].active )
   END_RUNG wire#w2
   RUNG wire#powerrail
      Contact( "SysDB_MP_Function_OP70".CycleType.Function[#t_Line].left )
      wire#w3
      S_SR(operand := "SysDB_MP_Function_OP70".CycleType.Function[#t_Line].active, r1 := wire#w4)
      wire#w5
      Coil( "AnwDB_StructureSelection_OP70".CycleType.Bypass_DamperCaps_FEED )
   END_RUNG
   RUNG wire#powerrail
      P_Contact(operand := "PunchSettings".Bypass.BypassDamperCapFeeding, bit := "GraDB2_FG01_Station_OP70".fpDamperCap_Feed_Deselection)
   END_RUNG wire#w3
   RUNG wire#powerrail
      Contact( "SysDB_MP_Function_OP70".CycleType.Function[#t_Line].right )
   END_RUNG wire#w4
   RUNG wire#powerrail
      N_Contact(operand := "PunchSettings".Bypass.BypassDamperCapFeeding, bit := "GraDB2_FG01_Station_OP70".fnDamperCap_Feed_Deselection)
   END_RUNG wire#w4
   RUNG wire#w5
      P_Trig( "AnwDB_StructureSelection_OP70".CycleType.fpBypass_DamperCaps_FEED )
      S_Coil( "PunchSettings".Bypass.BypassDamperCapFeeding )
   END_RUNG
   RUNG wire#w5
      N_Trig( "AnwDB_StructureSelection_OP70".CycleType.fnBypass_DamperCaps_FEED )
      R_Coil( "PunchSettings".Bypass.BypassDamperCapFeeding )
   END_RUNG
   // the same network as SCL:
   #t_Line := 4;
   "SysFC_HMI_Functions"("Type" := WSTRING#'"CycleType"',
                         Line := #t_Line,
                         "Enable Left" := #t_Enable_left,
                         "Enable Right" := #t_Enable_right,
                         "End Pos. Left" := "SysDB_MP_Function_OP70".CycleType.Function[#t_Line].active,
                         "End Pos. Right" := NOT "SysDB_MP_Function_OP70".CycleType.Function[#t_Line].active,
                         Position := 0.0,
                         "Hide Pos." := true,
                         "Hide Left Arrow" := false,
                         "Hide Right Arrow" := false,
                         LTLL_Config := "LTLL_Config".THIS[0],
                         LTLL_Data := "LTLL_Data".HMI[0],
                         Function_left => "SysDB_MP_Function_OP70".CycleType.Function[#t_Line].left,
                         Function_right => "SysDB_MP_Function_OP70".CycleType.Function[#t_Line].right,
                         ConfigFault => "SysDB_MP_Function_OP70".CycleType.Function[#t_Line].ConfigFault);
   #_w1 := "PunchSettings".Bypass.BypassDamperCapFeeding AND NOT "GraDB2_FG01_Station_OP70".fpDamperCap_Feed_Deselection;   // rising edge of "PunchSettings".Bypass.BypassDamperCapFeeding
   "GraDB2_FG01_Station_OP70".fpDamperCap_Feed_Deselection := "PunchSettings".Bypass.BypassDamperCapFeeding;
   #_w2 := NOT "PunchSettings".Bypass.BypassDamperCapFeeding AND "GraDB2_FG01_Station_OP70".fnDamperCap_Feed_Deselection;   // falling edge of "PunchSettings".Bypass.BypassDamperCapFeeding
   "GraDB2_FG01_Station_OP70".fnDamperCap_Feed_Deselection := "PunchSettings".Bypass.BypassDamperCapFeeding;
   #_w3 := "SysDB_MP_Function_OP70".CycleType.Function[#t_Line].right OR #_w2;
   IF "SysDB_MP_Function_OP70".CycleType.Function[#t_Line].left OR #_w1 THEN
       "SysDB_MP_Function_OP70".CycleType.Function[#t_Line].active := TRUE;   // SR flip-flop
   END_IF;
   IF #_w3 THEN "SysDB_MP_Function_OP70".CycleType.Function[#t_Line].active := FALSE; END_IF;
   "AnwDB_StructureSelection_OP70".CycleType.Bypass_DamperCaps_FEED := "SysDB_MP_Function_OP70".CycleType.Function[#t_Line].active;
   #_w4 := "SysDB_MP_Function_OP70".CycleType.Function[#t_Line].active AND NOT "AnwDB_StructureSelection_OP70".CycleType.fpBypass_DamperCaps_FEED;   // rising edge
   "AnwDB_StructureSelection_OP70".CycleType.fpBypass_DamperCaps_FEED := "SysDB_MP_Function_OP70".CycleType.Function[#t_Line].active;
   IF #_w4 THEN "PunchSettings".Bypass.BypassDamperCapFeeding := TRUE; END_IF;
   #_w5 := NOT "SysDB_MP_Function_OP70".CycleType.Function[#t_Line].active AND "AnwDB_StructureSelection_OP70".CycleType.fnBypass_DamperCaps_FEED;   // falling edge
   "AnwDB_StructureSelection_OP70".CycleType.fnBypass_DamperCaps_FEED := "SysDB_MP_Function_OP70".CycleType.Function[#t_Line].active;
   IF #_w5 THEN "PunchSettings".Bypass.BypassDamperCapFeeding := FALSE; END_IF;
END_REGION

REGION Network 18: CycleType - (line 5) - Damper Cap Camera Bypass
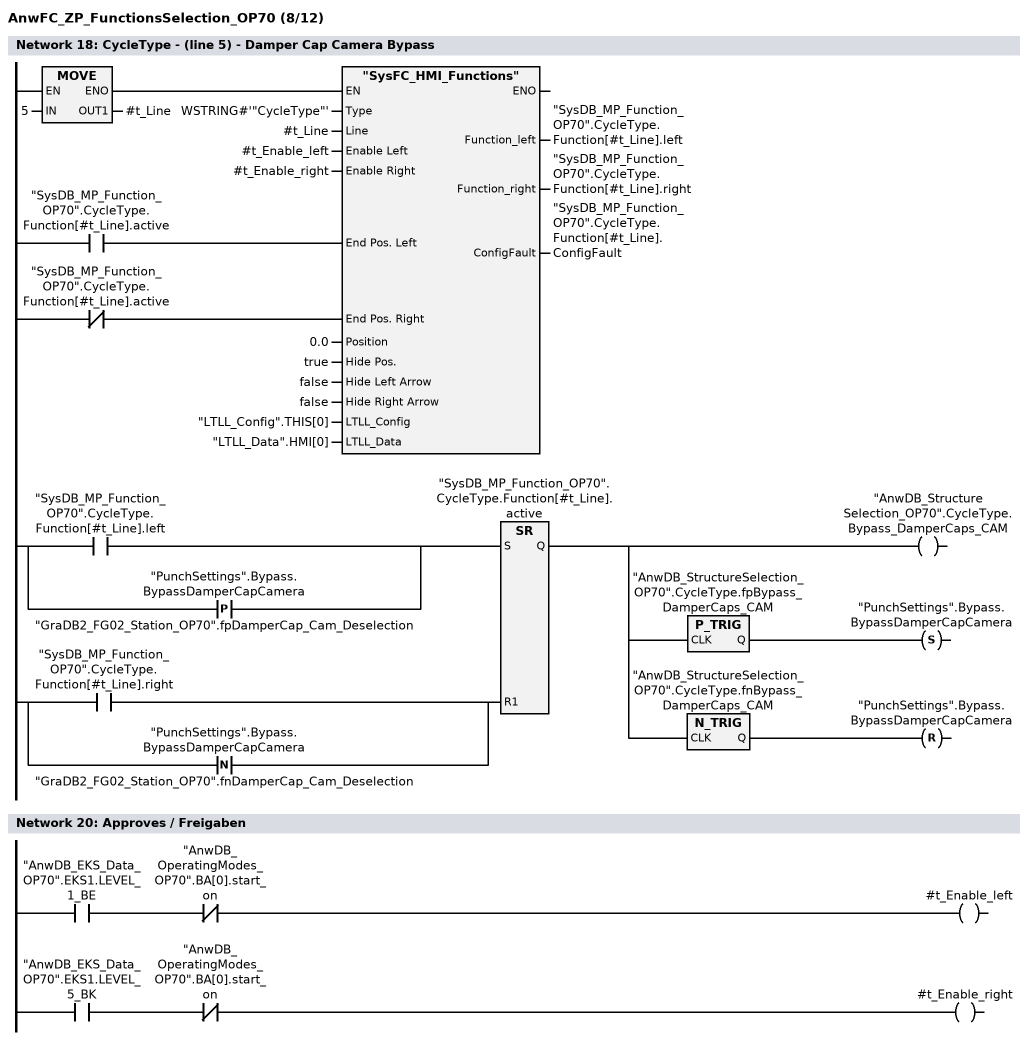
   RUNG wire#powerrail
      Move(in := 5, out1 => #t_Line)
      "SysFC_HMI_Functions"("End Pos. Left" := wire#w1, "End Pos. Right" := wire#w2, "Type" := WSTRING#'"CycleType"', Line := #t_Line, "Enable Left" := #t_Enable_left, "Enable Right" := #t_Enable_right, Position := 0.0, "Hide Pos." := true, "Hide Left Arrow" := false, "Hide Right Arrow" := false, LTLL_Config := "LTLL_Config".THIS[0], LTLL_Data := "LTLL_Data".HMI[0], Function_left => "SysDB_MP_Function_OP70".CycleType.Function[#t_Line].left, Function_right => "SysDB_MP_Function_OP70".CycleType.Function[#t_Line].right, ConfigFault => "SysDB_MP_Function_OP70".CycleType.Function[#t_Line].ConfigFault)
   END_RUNG
   RUNG wire#powerrail
      Contact( "SysDB_MP_Function_OP70".CycleType.Function[#t_Line].active )
   END_RUNG wire#w1
   RUNG wire#powerrail
      I_Contact( "SysDB_MP_Function_OP70".CycleType.Function[#t_Line].active )
   END_RUNG wire#w2
   RUNG wire#powerrail
      Contact( "SysDB_MP_Function_OP70".CycleType.Function[#t_Line].left )
      wire#w3
      S_SR(operand := "SysDB_MP_Function_OP70".CycleType.Function[#t_Line].active, r1 := wire#w4)
      wire#w5
      Coil( "AnwDB_StructureSelection_OP70".CycleType.Bypass_DamperCaps_CAM )
   END_RUNG
   RUNG wire#powerrail
      P_Contact(operand := "PunchSettings".Bypass.BypassDamperCapCamera, bit := "GraDB2_FG02_Station_OP70".fpDamperCap_Cam_Deselection)
   END_RUNG wire#w3
   RUNG wire#powerrail
      Contact( "SysDB_MP_Function_OP70".CycleType.Function[#t_Line].right )
   END_RUNG wire#w4
   RUNG wire#powerrail
      N_Contact(operand := "PunchSettings".Bypass.BypassDamperCapCamera, bit := "GraDB2_FG02_Station_OP70".fnDamperCap_Cam_Deselection)
   END_RUNG wire#w4
   RUNG wire#w5
      P_Trig( "AnwDB_StructureSelection_OP70".CycleType.fpBypass_DamperCaps_CAM )
      S_Coil( "PunchSettings".Bypass.BypassDamperCapCamera )
   END_RUNG
   RUNG wire#w5
      N_Trig( "AnwDB_StructureSelection_OP70".CycleType.fnBypass_DamperCaps_CAM )
      R_Coil( "PunchSettings".Bypass.BypassDamperCapCamera )
   END_RUNG
   // the same network as SCL:
   #t_Line := 5;
   "SysFC_HMI_Functions"("Type" := WSTRING#'"CycleType"',
                         Line := #t_Line,
                         "Enable Left" := #t_Enable_left,
                         "Enable Right" := #t_Enable_right,
                         "End Pos. Left" := "SysDB_MP_Function_OP70".CycleType.Function[#t_Line].active,
                         "End Pos. Right" := NOT "SysDB_MP_Function_OP70".CycleType.Function[#t_Line].active,
                         Position := 0.0,
                         "Hide Pos." := true,
                         "Hide Left Arrow" := false,
                         "Hide Right Arrow" := false,
                         LTLL_Config := "LTLL_Config".THIS[0],
                         LTLL_Data := "LTLL_Data".HMI[0],
                         Function_left => "SysDB_MP_Function_OP70".CycleType.Function[#t_Line].left,
                         Function_right => "SysDB_MP_Function_OP70".CycleType.Function[#t_Line].right,
                         ConfigFault => "SysDB_MP_Function_OP70".CycleType.Function[#t_Line].ConfigFault);
   #_w1 := "PunchSettings".Bypass.BypassDamperCapCamera AND NOT "GraDB2_FG02_Station_OP70".fpDamperCap_Cam_Deselection;   // rising edge of "PunchSettings".Bypass.BypassDamperCapCamera
   "GraDB2_FG02_Station_OP70".fpDamperCap_Cam_Deselection := "PunchSettings".Bypass.BypassDamperCapCamera;
   #_w2 := NOT "PunchSettings".Bypass.BypassDamperCapCamera AND "GraDB2_FG02_Station_OP70".fnDamperCap_Cam_Deselection;   // falling edge of "PunchSettings".Bypass.BypassDamperCapCamera
   "GraDB2_FG02_Station_OP70".fnDamperCap_Cam_Deselection := "PunchSettings".Bypass.BypassDamperCapCamera;
   #_w3 := "SysDB_MP_Function_OP70".CycleType.Function[#t_Line].right OR #_w2;
   IF "SysDB_MP_Function_OP70".CycleType.Function[#t_Line].left OR #_w1 THEN
       "SysDB_MP_Function_OP70".CycleType.Function[#t_Line].active := TRUE;   // SR flip-flop
   END_IF;
   IF #_w3 THEN "SysDB_MP_Function_OP70".CycleType.Function[#t_Line].active := FALSE; END_IF;
   "AnwDB_StructureSelection_OP70".CycleType.Bypass_DamperCaps_CAM := "SysDB_MP_Function_OP70".CycleType.Function[#t_Line].active;
   #_w4 := "SysDB_MP_Function_OP70".CycleType.Function[#t_Line].active AND NOT "AnwDB_StructureSelection_OP70".CycleType.fpBypass_DamperCaps_CAM;   // rising edge
   "AnwDB_StructureSelection_OP70".CycleType.fpBypass_DamperCaps_CAM := "SysDB_MP_Function_OP70".CycleType.Function[#t_Line].active;
   IF #_w4 THEN "PunchSettings".Bypass.BypassDamperCapCamera := TRUE; END_IF;
   #_w5 := NOT "SysDB_MP_Function_OP70".CycleType.Function[#t_Line].active AND "AnwDB_StructureSelection_OP70".CycleType.fnBypass_DamperCaps_CAM;   // falling edge
   "AnwDB_StructureSelection_OP70".CycleType.fnBypass_DamperCaps_CAM := "SysDB_MP_Function_OP70".CycleType.Function[#t_Line].active;
   IF #_w5 THEN "PunchSettings".Bypass.BypassDamperCapCamera := FALSE; END_IF;
END_REGION

REGION Network 19: ######## USER DEFINE ######### / ############ USER DEFINE ############
END_REGION

REGION Network 20: Approves / Freigaben
   RUNG wire#powerrail
      Contact( "AnwDB_EKS_Data_OP70".EKS1.LEVEL_1_BE )
      I_Contact( "AnwDB_OperatingModes_OP70".BA[0].start_on )
      Coil( #t_Enable_left )
   END_RUNG
   RUNG wire#powerrail
      Contact( "AnwDB_EKS_Data_OP70".EKS1.LEVEL_5_BK )
      I_Contact( "AnwDB_OperatingModes_OP70".BA[0].start_on )
      Coil( #t_Enable_right )
   END_RUNG
   // the same network as SCL:
   #t_Enable_left := "AnwDB_EKS_Data_OP70".EKS1.LEVEL_1_BE AND NOT "AnwDB_OperatingModes_OP70".BA[0].start_on;
   #t_Enable_right := "AnwDB_EKS_Data_OP70".EKS1.LEVEL_5_BK AND NOT "AnwDB_OperatingModes_OP70".BA[0].start_on;
END_REGION

REGION Network 21: Userdefine - (line 1) - IBM Modus / Userdefine - (Zeile 1) - IBM Modus
   // Valid types- WSTRING#'"Setup"';- WSTRING#'"PowerUp"';- WSTRING#'"Unit"';- WSTRING#'"NutRunner"';- WSTRING#'"NutRunnerGroup"';- WSTRING#'"CycleType"';- WSTRING#'"UserDefine"';
   // Gültige Typen
   // - WSTRING#'"Setup"'
   // - WSTRING#'"PowerUp"'
   // - WSTRING#'"Unit"'
   // - WSTRING#'"NutRunner"'
   // - WSTRING#'"NutRunnerGroup"'
   // - WSTRING#'"CycleType"'
   // - WSTRING#'"UserDefine"'
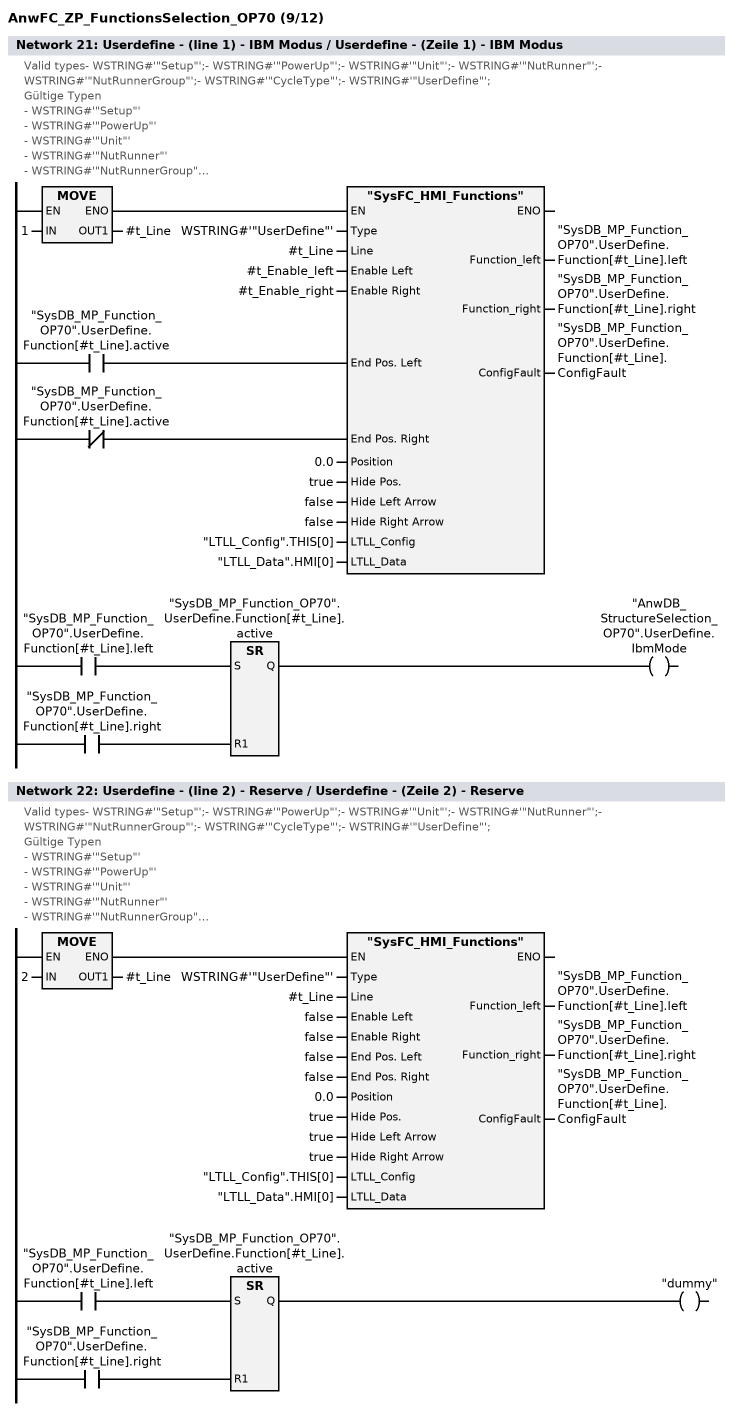
   RUNG wire#powerrail
      Move(in := 1, out1 => #t_Line)
      "SysFC_HMI_Functions"("End Pos. Left" := wire#w1, "End Pos. Right" := wire#w2, "Type" := WSTRING#'"UserDefine"', Line := #t_Line, "Enable Left" := #t_Enable_left, "Enable Right" := #t_Enable_right, Position := 0.0, "Hide Pos." := true, "Hide Left Arrow" := false, "Hide Right Arrow" := false, LTLL_Config := "LTLL_Config".THIS[0], LTLL_Data := "LTLL_Data".HMI[0], Function_left => "SysDB_MP_Function_OP70".UserDefine.Function[#t_Line].left, Function_right => "SysDB_MP_Function_OP70".UserDefine.Function[#t_Line].right, ConfigFault => "SysDB_MP_Function_OP70".UserDefine.Function[#t_Line].ConfigFault)
   END_RUNG
   RUNG wire#powerrail
      Contact( "SysDB_MP_Function_OP70".UserDefine.Function[#t_Line].active )
   END_RUNG wire#w1
   RUNG wire#powerrail
      I_Contact( "SysDB_MP_Function_OP70".UserDefine.Function[#t_Line].active )
   END_RUNG wire#w2
   RUNG wire#powerrail
      Contact( "SysDB_MP_Function_OP70".UserDefine.Function[#t_Line].left )
      S_SR(operand := "SysDB_MP_Function_OP70".UserDefine.Function[#t_Line].active, r1 := wire#w3)
      Coil( "AnwDB_StructureSelection_OP70".UserDefine.IbmMode )
   END_RUNG
   RUNG wire#powerrail
      Contact( "SysDB_MP_Function_OP70".UserDefine.Function[#t_Line].right )
   END_RUNG wire#w3
   // the same network as SCL:
   #t_Line := 1;
   "SysFC_HMI_Functions"("Type" := WSTRING#'"UserDefine"',
                         Line := #t_Line,
                         "Enable Left" := #t_Enable_left,
                         "Enable Right" := #t_Enable_right,
                         "End Pos. Left" := "SysDB_MP_Function_OP70".UserDefine.Function[#t_Line].active,
                         "End Pos. Right" := NOT "SysDB_MP_Function_OP70".UserDefine.Function[#t_Line].active,
                         Position := 0.0,
                         "Hide Pos." := true,
                         "Hide Left Arrow" := false,
                         "Hide Right Arrow" := false,
                         LTLL_Config := "LTLL_Config".THIS[0],
                         LTLL_Data := "LTLL_Data".HMI[0],
                         Function_left => "SysDB_MP_Function_OP70".UserDefine.Function[#t_Line].left,
                         Function_right => "SysDB_MP_Function_OP70".UserDefine.Function[#t_Line].right,
                         ConfigFault => "SysDB_MP_Function_OP70".UserDefine.Function[#t_Line].ConfigFault);
   #_w1 := "SysDB_MP_Function_OP70".UserDefine.Function[#t_Line].right;
   IF "SysDB_MP_Function_OP70".UserDefine.Function[#t_Line].left THEN
       "SysDB_MP_Function_OP70".UserDefine.Function[#t_Line].active := TRUE;   // SR flip-flop
   END_IF;
   IF #_w1 THEN "SysDB_MP_Function_OP70".UserDefine.Function[#t_Line].active := FALSE; END_IF;
   "AnwDB_StructureSelection_OP70".UserDefine.IbmMode := "SysDB_MP_Function_OP70".UserDefine.Function[#t_Line].active;
END_REGION

REGION Network 22: Userdefine - (line 2) - Reserve / Userdefine - (Zeile 2) - Reserve
   // Valid types- WSTRING#'"Setup"';- WSTRING#'"PowerUp"';- WSTRING#'"Unit"';- WSTRING#'"NutRunner"';- WSTRING#'"NutRunnerGroup"';- WSTRING#'"CycleType"';- WSTRING#'"UserDefine"';
   // Gültige Typen
   // - WSTRING#'"Setup"'
   // - WSTRING#'"PowerUp"'
   // - WSTRING#'"Unit"'
   // - WSTRING#'"NutRunner"'
   // - WSTRING#'"NutRunnerGroup"'
   // - WSTRING#'"CycleType"'
   // - WSTRING#'"UserDefine"'
   RUNG wire#powerrail
      Move(in := 2, out1 => #t_Line)
      "SysFC_HMI_Functions"("Type" := WSTRING#'"UserDefine"', Line := #t_Line, "Enable Left" := false, "Enable Right" := false, "End Pos. Left" := false, "End Pos. Right" := false, Position := 0.0, "Hide Pos." := true, "Hide Left Arrow" := true, "Hide Right Arrow" := true, LTLL_Config := "LTLL_Config".THIS[0], LTLL_Data := "LTLL_Data".HMI[0], Function_left => "SysDB_MP_Function_OP70".UserDefine.Function[#t_Line].left, Function_right => "SysDB_MP_Function_OP70".UserDefine.Function[#t_Line].right, ConfigFault => "SysDB_MP_Function_OP70".UserDefine.Function[#t_Line].ConfigFault)
   END_RUNG
   RUNG wire#powerrail
      Contact( "SysDB_MP_Function_OP70".UserDefine.Function[#t_Line].left )
      S_SR(operand := "SysDB_MP_Function_OP70".UserDefine.Function[#t_Line].active, r1 := wire#w1)
      Coil( "dummy" )
   END_RUNG
   RUNG wire#powerrail
      Contact( "SysDB_MP_Function_OP70".UserDefine.Function[#t_Line].right )
   END_RUNG wire#w1
   // the same network as SCL:
   #t_Line := 2;
   "SysFC_HMI_Functions"("Type" := WSTRING#'"UserDefine"',
                         Line := #t_Line,
                         "Enable Left" := false,
                         "Enable Right" := false,
                         "End Pos. Left" := false,
                         "End Pos. Right" := false,
                         Position := 0.0,
                         "Hide Pos." := true,
                         "Hide Left Arrow" := true,
                         "Hide Right Arrow" := true,
                         LTLL_Config := "LTLL_Config".THIS[0],
                         LTLL_Data := "LTLL_Data".HMI[0],
                         Function_left => "SysDB_MP_Function_OP70".UserDefine.Function[#t_Line].left,
                         Function_right => "SysDB_MP_Function_OP70".UserDefine.Function[#t_Line].right,
                         ConfigFault => "SysDB_MP_Function_OP70".UserDefine.Function[#t_Line].ConfigFault);
   #_w1 := "SysDB_MP_Function_OP70".UserDefine.Function[#t_Line].right;
   IF "SysDB_MP_Function_OP70".UserDefine.Function[#t_Line].left THEN
       "SysDB_MP_Function_OP70".UserDefine.Function[#t_Line].active := TRUE;   // SR flip-flop
   END_IF;
   IF #_w1 THEN "SysDB_MP_Function_OP70".UserDefine.Function[#t_Line].active := FALSE; END_IF;
   "dummy" := "SysDB_MP_Function_OP70".UserDefine.Function[#t_Line].active;
END_REGION

REGION Network 23: Userdefine - (line 3) - Reserve / Userdefine - (Zeile 3) - Reserve
   // Valid types- WSTRING#'"Setup"';- WSTRING#'"PowerUp"';- WSTRING#'"Unit"';- WSTRING#'"NutRunner"';- WSTRING#'"NutRunnerGroup"';- WSTRING#'"CycleType"';- WSTRING#'"UserDefine"';
   // Gültige Typen
   // - WSTRING#'"Setup"'
   // - WSTRING#'"PowerUp"'
   // - WSTRING#'"Unit"'
   // - WSTRING#'"NutRunner"'
   // - WSTRING#'"NutRunnerGroup"'
   // - WSTRING#'"CycleType"'
   // - WSTRING#'"UserDefine"'
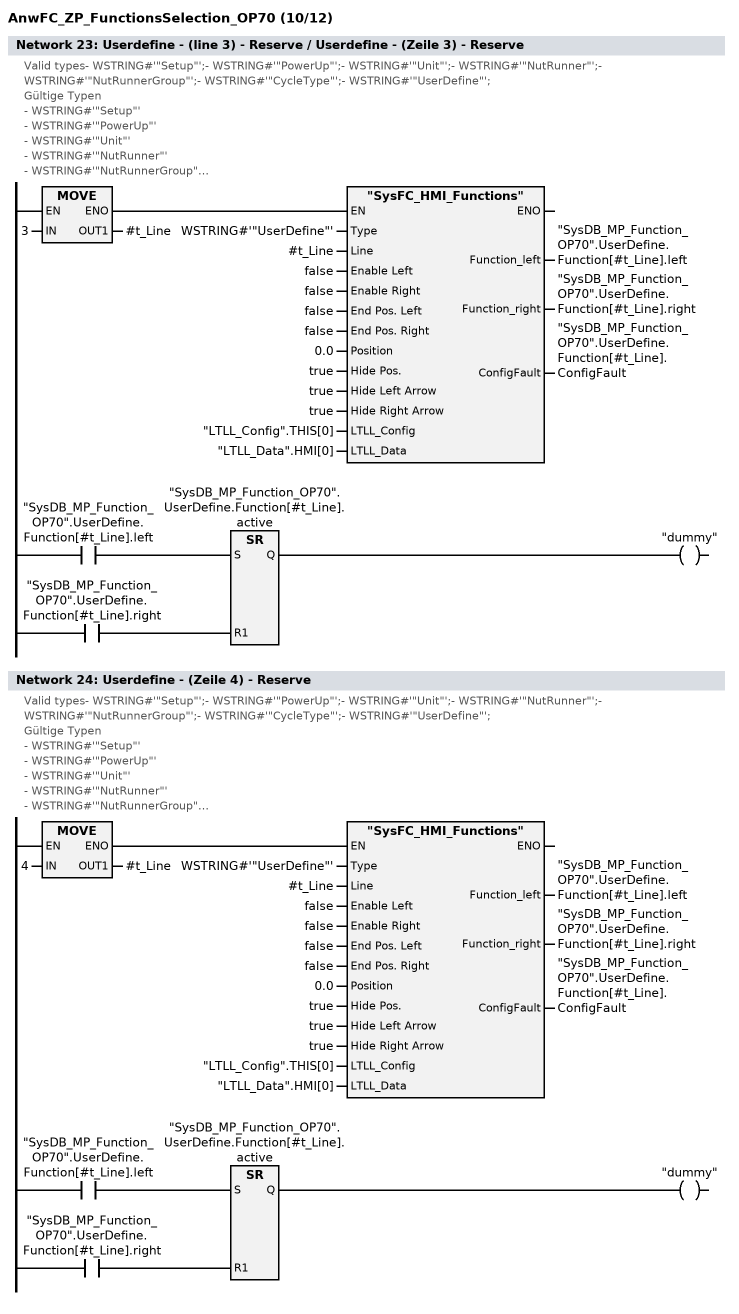
   RUNG wire#powerrail
      Move(in := 3, out1 => #t_Line)
      "SysFC_HMI_Functions"("Type" := WSTRING#'"UserDefine"', Line := #t_Line, "Enable Left" := false, "Enable Right" := false, "End Pos. Left" := false, "End Pos. Right" := false, Position := 0.0, "Hide Pos." := true, "Hide Left Arrow" := true, "Hide Right Arrow" := true, LTLL_Config := "LTLL_Config".THIS[0], LTLL_Data := "LTLL_Data".HMI[0], Function_left => "SysDB_MP_Function_OP70".UserDefine.Function[#t_Line].left, Function_right => "SysDB_MP_Function_OP70".UserDefine.Function[#t_Line].right, ConfigFault => "SysDB_MP_Function_OP70".UserDefine.Function[#t_Line].ConfigFault)
   END_RUNG
   RUNG wire#powerrail
      Contact( "SysDB_MP_Function_OP70".UserDefine.Function[#t_Line].left )
      S_SR(operand := "SysDB_MP_Function_OP70".UserDefine.Function[#t_Line].active, r1 := wire#w1)
      Coil( "dummy" )
   END_RUNG
   RUNG wire#powerrail
      Contact( "SysDB_MP_Function_OP70".UserDefine.Function[#t_Line].right )
   END_RUNG wire#w1
   // the same network as SCL:
   #t_Line := 3;
   "SysFC_HMI_Functions"("Type" := WSTRING#'"UserDefine"',
                         Line := #t_Line,
                         "Enable Left" := false,
                         "Enable Right" := false,
                         "End Pos. Left" := false,
                         "End Pos. Right" := false,
                         Position := 0.0,
                         "Hide Pos." := true,
                         "Hide Left Arrow" := true,
                         "Hide Right Arrow" := true,
                         LTLL_Config := "LTLL_Config".THIS[0],
                         LTLL_Data := "LTLL_Data".HMI[0],
                         Function_left => "SysDB_MP_Function_OP70".UserDefine.Function[#t_Line].left,
                         Function_right => "SysDB_MP_Function_OP70".UserDefine.Function[#t_Line].right,
                         ConfigFault => "SysDB_MP_Function_OP70".UserDefine.Function[#t_Line].ConfigFault);
   #_w1 := "SysDB_MP_Function_OP70".UserDefine.Function[#t_Line].right;
   IF "SysDB_MP_Function_OP70".UserDefine.Function[#t_Line].left THEN
       "SysDB_MP_Function_OP70".UserDefine.Function[#t_Line].active := TRUE;   // SR flip-flop
   END_IF;
   IF #_w1 THEN "SysDB_MP_Function_OP70".UserDefine.Function[#t_Line].active := FALSE; END_IF;
   "dummy" := "SysDB_MP_Function_OP70".UserDefine.Function[#t_Line].active;
END_REGION

REGION Network 24: Userdefine - (Zeile 4) - Reserve
   // Valid types- WSTRING#'"Setup"';- WSTRING#'"PowerUp"';- WSTRING#'"Unit"';- WSTRING#'"NutRunner"';- WSTRING#'"NutRunnerGroup"';- WSTRING#'"CycleType"';- WSTRING#'"UserDefine"';
   // Gültige Typen
   // - WSTRING#'"Setup"'
   // - WSTRING#'"PowerUp"'
   // - WSTRING#'"Unit"'
   // - WSTRING#'"NutRunner"'
   // - WSTRING#'"NutRunnerGroup"'
   // - WSTRING#'"CycleType"'
   // - WSTRING#'"UserDefine"'
   RUNG wire#powerrail
      Move(in := 4, out1 => #t_Line)
      "SysFC_HMI_Functions"("Type" := WSTRING#'"UserDefine"', Line := #t_Line, "Enable Left" := false, "Enable Right" := false, "End Pos. Left" := false, "End Pos. Right" := false, Position := 0.0, "Hide Pos." := true, "Hide Left Arrow" := true, "Hide Right Arrow" := true, LTLL_Config := "LTLL_Config".THIS[0], LTLL_Data := "LTLL_Data".HMI[0], Function_left => "SysDB_MP_Function_OP70".UserDefine.Function[#t_Line].left, Function_right => "SysDB_MP_Function_OP70".UserDefine.Function[#t_Line].right, ConfigFault => "SysDB_MP_Function_OP70".UserDefine.Function[#t_Line].ConfigFault)
   END_RUNG
   RUNG wire#powerrail
      Contact( "SysDB_MP_Function_OP70".UserDefine.Function[#t_Line].left )
      S_SR(operand := "SysDB_MP_Function_OP70".UserDefine.Function[#t_Line].active, r1 := wire#w1)
      Coil( "dummy" )
   END_RUNG
   RUNG wire#powerrail
      Contact( "SysDB_MP_Function_OP70".UserDefine.Function[#t_Line].right )
   END_RUNG wire#w1
   // the same network as SCL:
   #t_Line := 4;
   "SysFC_HMI_Functions"("Type" := WSTRING#'"UserDefine"',
                         Line := #t_Line,
                         "Enable Left" := false,
                         "Enable Right" := false,
                         "End Pos. Left" := false,
                         "End Pos. Right" := false,
                         Position := 0.0,
                         "Hide Pos." := true,
                         "Hide Left Arrow" := true,
                         "Hide Right Arrow" := true,
                         LTLL_Config := "LTLL_Config".THIS[0],
                         LTLL_Data := "LTLL_Data".HMI[0],
                         Function_left => "SysDB_MP_Function_OP70".UserDefine.Function[#t_Line].left,
                         Function_right => "SysDB_MP_Function_OP70".UserDefine.Function[#t_Line].right,
                         ConfigFault => "SysDB_MP_Function_OP70".UserDefine.Function[#t_Line].ConfigFault);
   #_w1 := "SysDB_MP_Function_OP70".UserDefine.Function[#t_Line].right;
   IF "SysDB_MP_Function_OP70".UserDefine.Function[#t_Line].left THEN
       "SysDB_MP_Function_OP70".UserDefine.Function[#t_Line].active := TRUE;   // SR flip-flop
   END_IF;
   IF #_w1 THEN "SysDB_MP_Function_OP70".UserDefine.Function[#t_Line].active := FALSE; END_IF;
   "dummy" := "SysDB_MP_Function_OP70".UserDefine.Function[#t_Line].active;
END_REGION

REGION Network 25: Userdefine - (Zeile 5) - Reserve
   // Valid types- WSTRING#'"Setup"';- WSTRING#'"PowerUp"';- WSTRING#'"Unit"';- WSTRING#'"NutRunner"';- WSTRING#'"NutRunnerGroup"';- WSTRING#'"CycleType"';- WSTRING#'"UserDefine"';
   // Gültige Typen
   // - WSTRING#'"Setup"'
   // - WSTRING#'"PowerUp"'
   // - WSTRING#'"Unit"'
   // - WSTRING#'"NutRunner"'
   // - WSTRING#'"NutRunnerGroup"'
   // - WSTRING#'"CycleType"'
   // - WSTRING#'"UserDefine"'
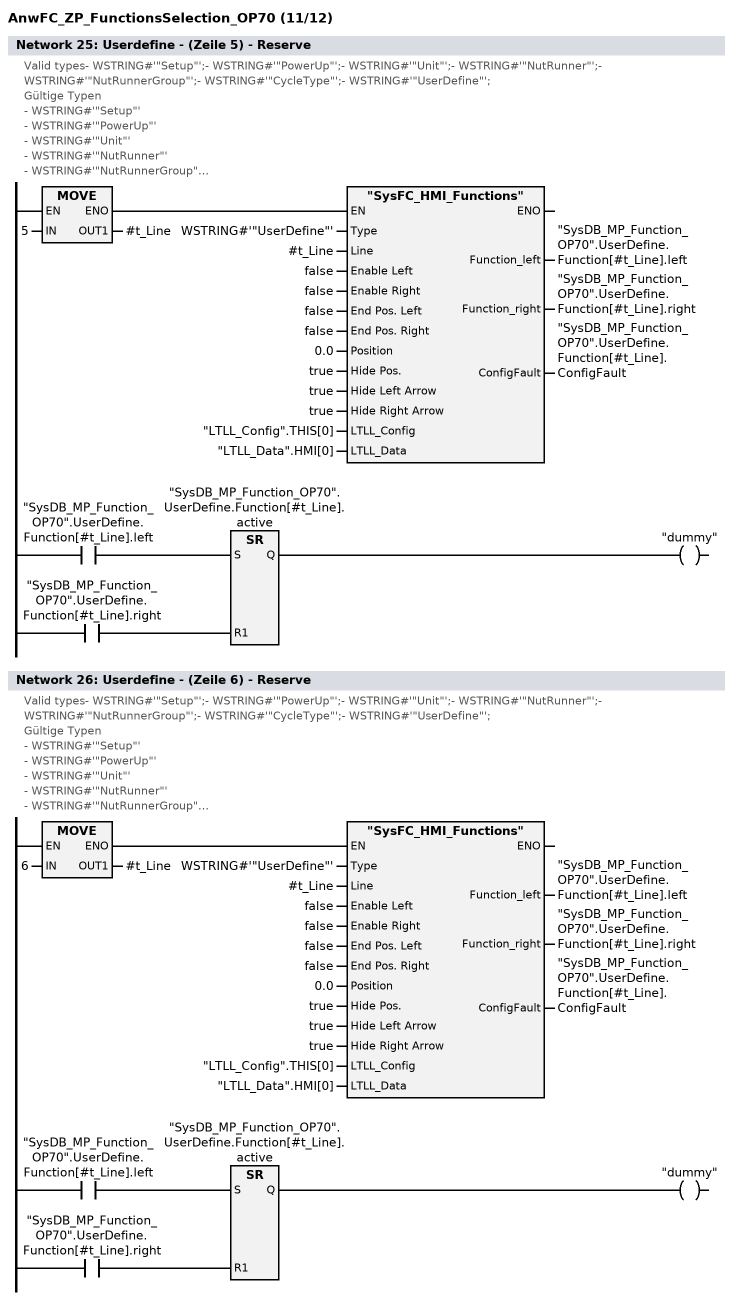
   RUNG wire#powerrail
      Move(in := 5, out1 => #t_Line)
      "SysFC_HMI_Functions"("Type" := WSTRING#'"UserDefine"', Line := #t_Line, "Enable Left" := false, "Enable Right" := false, "End Pos. Left" := false, "End Pos. Right" := false, Position := 0.0, "Hide Pos." := true, "Hide Left Arrow" := true, "Hide Right Arrow" := true, LTLL_Config := "LTLL_Config".THIS[0], LTLL_Data := "LTLL_Data".HMI[0], Function_left => "SysDB_MP_Function_OP70".UserDefine.Function[#t_Line].left, Function_right => "SysDB_MP_Function_OP70".UserDefine.Function[#t_Line].right, ConfigFault => "SysDB_MP_Function_OP70".UserDefine.Function[#t_Line].ConfigFault)
   END_RUNG
   RUNG wire#powerrail
      Contact( "SysDB_MP_Function_OP70".UserDefine.Function[#t_Line].left )
      S_SR(operand := "SysDB_MP_Function_OP70".UserDefine.Function[#t_Line].active, r1 := wire#w1)
      Coil( "dummy" )
   END_RUNG
   RUNG wire#powerrail
      Contact( "SysDB_MP_Function_OP70".UserDefine.Function[#t_Line].right )
   END_RUNG wire#w1
   // the same network as SCL:
   #t_Line := 5;
   "SysFC_HMI_Functions"("Type" := WSTRING#'"UserDefine"',
                         Line := #t_Line,
                         "Enable Left" := false,
                         "Enable Right" := false,
                         "End Pos. Left" := false,
                         "End Pos. Right" := false,
                         Position := 0.0,
                         "Hide Pos." := true,
                         "Hide Left Arrow" := true,
                         "Hide Right Arrow" := true,
                         LTLL_Config := "LTLL_Config".THIS[0],
                         LTLL_Data := "LTLL_Data".HMI[0],
                         Function_left => "SysDB_MP_Function_OP70".UserDefine.Function[#t_Line].left,
                         Function_right => "SysDB_MP_Function_OP70".UserDefine.Function[#t_Line].right,
                         ConfigFault => "SysDB_MP_Function_OP70".UserDefine.Function[#t_Line].ConfigFault);
   #_w1 := "SysDB_MP_Function_OP70".UserDefine.Function[#t_Line].right;
   IF "SysDB_MP_Function_OP70".UserDefine.Function[#t_Line].left THEN
       "SysDB_MP_Function_OP70".UserDefine.Function[#t_Line].active := TRUE;   // SR flip-flop
   END_IF;
   IF #_w1 THEN "SysDB_MP_Function_OP70".UserDefine.Function[#t_Line].active := FALSE; END_IF;
   "dummy" := "SysDB_MP_Function_OP70".UserDefine.Function[#t_Line].active;
END_REGION

REGION Network 26: Userdefine - (Zeile 6) - Reserve
   // Valid types- WSTRING#'"Setup"';- WSTRING#'"PowerUp"';- WSTRING#'"Unit"';- WSTRING#'"NutRunner"';- WSTRING#'"NutRunnerGroup"';- WSTRING#'"CycleType"';- WSTRING#'"UserDefine"';
   // Gültige Typen
   // - WSTRING#'"Setup"'
   // - WSTRING#'"PowerUp"'
   // - WSTRING#'"Unit"'
   // - WSTRING#'"NutRunner"'
   // - WSTRING#'"NutRunnerGroup"'
   // - WSTRING#'"CycleType"'
   // - WSTRING#'"UserDefine"'
   RUNG wire#powerrail
      Move(in := 6, out1 => #t_Line)
      "SysFC_HMI_Functions"("Type" := WSTRING#'"UserDefine"', Line := #t_Line, "Enable Left" := false, "Enable Right" := false, "End Pos. Left" := false, "End Pos. Right" := false, Position := 0.0, "Hide Pos." := true, "Hide Left Arrow" := true, "Hide Right Arrow" := true, LTLL_Config := "LTLL_Config".THIS[0], LTLL_Data := "LTLL_Data".HMI[0], Function_left => "SysDB_MP_Function_OP70".UserDefine.Function[#t_Line].left, Function_right => "SysDB_MP_Function_OP70".UserDefine.Function[#t_Line].right, ConfigFault => "SysDB_MP_Function_OP70".UserDefine.Function[#t_Line].ConfigFault)
   END_RUNG
   RUNG wire#powerrail
      Contact( "SysDB_MP_Function_OP70".UserDefine.Function[#t_Line].left )
      S_SR(operand := "SysDB_MP_Function_OP70".UserDefine.Function[#t_Line].active, r1 := wire#w1)
      Coil( "dummy" )
   END_RUNG
   RUNG wire#powerrail
      Contact( "SysDB_MP_Function_OP70".UserDefine.Function[#t_Line].right )
   END_RUNG wire#w1
   // the same network as SCL:
   #t_Line := 6;
   "SysFC_HMI_Functions"("Type" := WSTRING#'"UserDefine"',
                         Line := #t_Line,
                         "Enable Left" := false,
                         "Enable Right" := false,
                         "End Pos. Left" := false,
                         "End Pos. Right" := false,
                         Position := 0.0,
                         "Hide Pos." := true,
                         "Hide Left Arrow" := true,
                         "Hide Right Arrow" := true,
                         LTLL_Config := "LTLL_Config".THIS[0],
                         LTLL_Data := "LTLL_Data".HMI[0],
                         Function_left => "SysDB_MP_Function_OP70".UserDefine.Function[#t_Line].left,
                         Function_right => "SysDB_MP_Function_OP70".UserDefine.Function[#t_Line].right,
                         ConfigFault => "SysDB_MP_Function_OP70".UserDefine.Function[#t_Line].ConfigFault);
   #_w1 := "SysDB_MP_Function_OP70".UserDefine.Function[#t_Line].right;
   IF "SysDB_MP_Function_OP70".UserDefine.Function[#t_Line].left THEN
       "SysDB_MP_Function_OP70".UserDefine.Function[#t_Line].active := TRUE;   // SR flip-flop
   END_IF;
   IF #_w1 THEN "SysDB_MP_Function_OP70".UserDefine.Function[#t_Line].active := FALSE; END_IF;
   "dummy" := "SysDB_MP_Function_OP70".UserDefine.Function[#t_Line].active;
END_REGION

REGION Network 27: ######## CHECKING OUT ######### / ############### AUSWERTUNG ###############
END_REGION

REGION Network 28: Deselection active / Abwahl aktiv
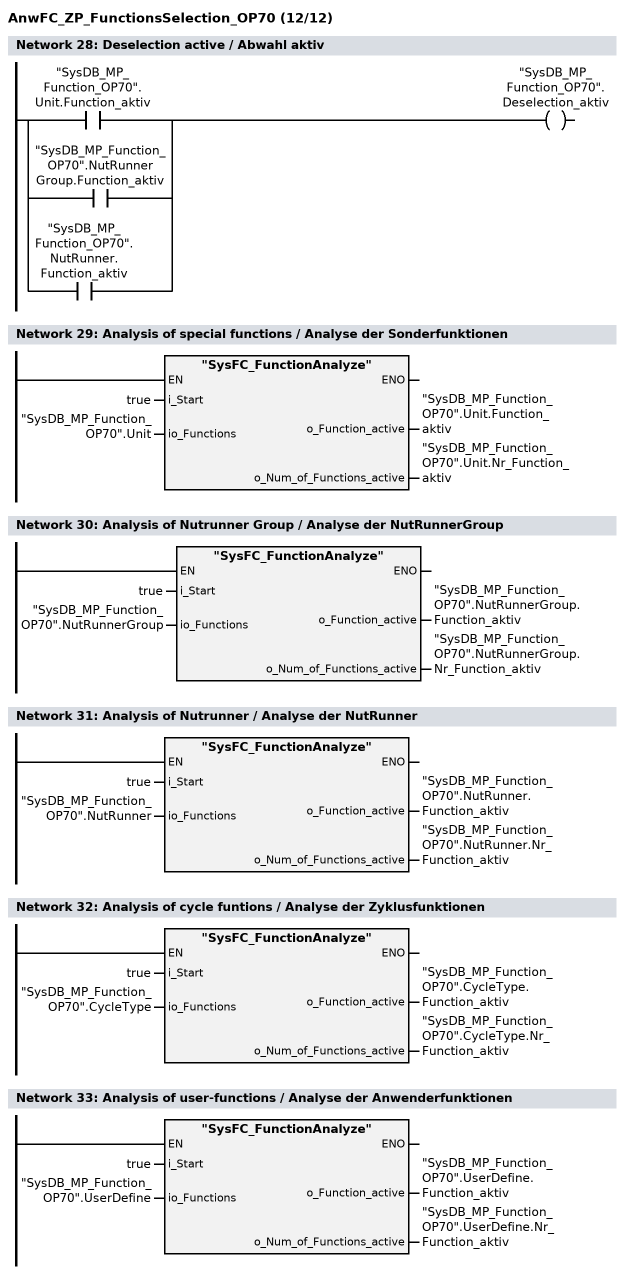
   RUNG wire#powerrail
      Contact( "SysDB_MP_Function_OP70".Unit.Function_aktiv )
      wire#w1
      Coil( "SysDB_MP_Function_OP70".Deselection_aktiv )
   END_RUNG
   RUNG wire#powerrail
      Contact( "SysDB_MP_Function_OP70".NutRunnerGroup.Function_aktiv )
   END_RUNG wire#w1
   RUNG wire#powerrail
      Contact( "SysDB_MP_Function_OP70".NutRunner.Function_aktiv )
   END_RUNG wire#w1
   // the same network as SCL:
   "SysDB_MP_Function_OP70".Deselection_aktiv := "SysDB_MP_Function_OP70".Unit.Function_aktiv OR "SysDB_MP_Function_OP70".NutRunnerGroup.Function_aktiv OR "SysDB_MP_Function_OP70".NutRunner.Function_aktiv;
END_REGION

REGION Network 29: Analysis of special functions / Analyse der Sonderfunktionen
   RUNG wire#powerrail
      "SysFC_FunctionAnalyze"(i_Start := true, io_Functions := "SysDB_MP_Function_OP70".Unit, o_Function_active => "SysDB_MP_Function_OP70".Unit.Function_aktiv, o_Num_of_Functions_active => "SysDB_MP_Function_OP70".Unit.Nr_Function_aktiv)
   END_RUNG
   // the same network as SCL:
   "SysFC_FunctionAnalyze"(i_Start := true,
                           io_Functions := "SysDB_MP_Function_OP70".Unit,
                           o_Function_active => "SysDB_MP_Function_OP70".Unit.Function_aktiv,
                           o_Num_of_Functions_active => "SysDB_MP_Function_OP70".Unit.Nr_Function_aktiv);
END_REGION

REGION Network 30: Analysis of Nutrunner Group / Analyse der NutRunnerGroup
   RUNG wire#powerrail
      "SysFC_FunctionAnalyze"(i_Start := true, io_Functions := "SysDB_MP_Function_OP70".NutRunnerGroup, o_Function_active => "SysDB_MP_Function_OP70".NutRunnerGroup.Function_aktiv, o_Num_of_Functions_active => "SysDB_MP_Function_OP70".NutRunnerGroup.Nr_Function_aktiv)
   END_RUNG
   // the same network as SCL:
   "SysFC_FunctionAnalyze"(i_Start := true,
                           io_Functions := "SysDB_MP_Function_OP70".NutRunnerGroup,
                           o_Function_active => "SysDB_MP_Function_OP70".NutRunnerGroup.Function_aktiv,
                           o_Num_of_Functions_active => "SysDB_MP_Function_OP70".NutRunnerGroup.Nr_Function_aktiv);
END_REGION

REGION Network 31: Analysis of Nutrunner / Analyse der NutRunner
   RUNG wire#powerrail
      "SysFC_FunctionAnalyze"(i_Start := true, io_Functions := "SysDB_MP_Function_OP70".NutRunner, o_Function_active => "SysDB_MP_Function_OP70".NutRunner.Function_aktiv, o_Num_of_Functions_active => "SysDB_MP_Function_OP70".NutRunner.Nr_Function_aktiv)
   END_RUNG
   // the same network as SCL:
   "SysFC_FunctionAnalyze"(i_Start := true,
                           io_Functions := "SysDB_MP_Function_OP70".NutRunner,
                           o_Function_active => "SysDB_MP_Function_OP70".NutRunner.Function_aktiv,
                           o_Num_of_Functions_active => "SysDB_MP_Function_OP70".NutRunner.Nr_Function_aktiv);
END_REGION

REGION Network 32: Analysis of cycle funtions / Analyse der Zyklusfunktionen
   RUNG wire#powerrail
      "SysFC_FunctionAnalyze"(i_Start := true, io_Functions := "SysDB_MP_Function_OP70".CycleType, o_Function_active => "SysDB_MP_Function_OP70".CycleType.Function_aktiv, o_Num_of_Functions_active => "SysDB_MP_Function_OP70".CycleType.Nr_Function_aktiv)
   END_RUNG
   // the same network as SCL:
   "SysFC_FunctionAnalyze"(i_Start := true,
                           io_Functions := "SysDB_MP_Function_OP70".CycleType,
                           o_Function_active => "SysDB_MP_Function_OP70".CycleType.Function_aktiv,
                           o_Num_of_Functions_active => "SysDB_MP_Function_OP70".CycleType.Nr_Function_aktiv);
END_REGION

REGION Network 33: Analysis of user-functions / Analyse der Anwenderfunktionen
   RUNG wire#powerrail
      "SysFC_FunctionAnalyze"(i_Start := true, io_Functions := "SysDB_MP_Function_OP70".UserDefine, o_Function_active => "SysDB_MP_Function_OP70".UserDefine.Function_aktiv, o_Num_of_Functions_active => "SysDB_MP_Function_OP70".UserDefine.Nr_Function_aktiv)
   END_RUNG
   // the same network as SCL:
   "SysFC_FunctionAnalyze"(i_Start := true,
                           io_Functions := "SysDB_MP_Function_OP70".UserDefine,
                           o_Function_active => "SysDB_MP_Function_OP70".UserDefine.Function_aktiv,
                           o_Num_of_Functions_active => "SysDB_MP_Function_OP70".UserDefine.Nr_Function_aktiv);
END_REGION
END_FUNCTION
